(* CODESYS project oscat311.library
   Company: OSCAT
   Version: 3.11
   Author: www.oscat.de
   Title: LIBRARY

Project tree, tasks and I/O mapping:
  libraries: Standard, 3.3.1.10 (System)
  Data types/
    data type CALENDAR
    data type COMPLEX
    data type CONSTANTS_LANGUAGE
    data type CONSTANTS_LOCATION
    data type CONSTANTS_MATH
    data type CONSTANTS_PHYS
    data type CONSTANTS_SETUP
    data type ESR_DATA
    data type HOLIDAY_DATA
    data type NETWORK_BUFFER
    data type NETWORK_BUFFER_SHORT
    data type NW_BUF_LONG
    data type NW_BUF_SHORT
    data type REAL2
    data type SDT
    data type TIMER_EVENT
    data type URL
    data type VECTOR_3
  Global Variables/
    global variables Constants
    global variables Globale_Variablen
    global variables Setup_Data
  POUs/
    Buffer Management/
      function _BUFFER_CLEAR [ST]
      function _BUFFER_INIT [ST]
      function _BUFFER_INSERT [ST]
      function _STRING_TO_BUFFER [ST]
      function BUFFER_COMP [ST]
      function BUFFER_SEARCH [ST]
      function BUFFER_TO_STRING [ST]
    Building/
      actuators/
        function block ACTUATOR_2P [ST]
        function block ACTUATOR_3P [ST]
        function block ACTUATOR_A [ST]
        function block ACTUATOR_COIL [ST]
        function block ACTUATOR_PUMP [ST]
        function block ACTUATOR_UD [ST]
        function block AUTORUN [ST]
      electrical/
        function block CLICK [ST]
        function block CLICK_MODE [ST]
        function block DEBOUNCE [ST]
        function block DIMM_2 [ST]
        function block DIMM_I [ST]
        function block F_LAMP [ST]
        function block PULSE_LENGTH [ST]
        function block PULSE_T [ST]
        function block SW_RECONFIG [ST]
        function block SWITCH_I [ST]
        function block SWITCH_X [ST]
        function block TIMER_1 [ST]
        function block TIMER_2 [ST]
        function TIMER_EVENT_DECODE [ST]
        function block TIMER_EXT [ST]
        function block TIMER_P4 [ST]
      HLK/
        function AIR_DENSITY [ST]
        function AIR_ENTHALPY [ST]
        function block BOILER [ST]
        function block BURNER [ST]
        function DEW_CON [ST]
        function DEW_RH [ST]
        function DEW_TEMP [ST]
        function HEAT_INDEX [ST]
        function block HEAT_METER [ST]
        function block HEAT_TEMP [ST]
        function block LEGIONELLA [ST]
        function SDD [ST]
        function SDD_NH3 [ST]
        function SDT_NH3 [ST]
        function block T_AVG24 [ST]
        function block TEMP_EXT [ST]
        function WATER_CP [ST]
        function WATER_DENSITY [ST]
        function WATER_ENTHALPY [ST]
        function WCT [ST]
      Jalousie/
        function block BLIND_ACTUATOR [ST]
        function block BLIND_CONTROL [ST]
        function block BLIND_CONTROL_S [ST]
        function block BLIND_INPUT [ST]
        function block BLIND_NIGHT [ST]
        function block BLIND_SCENE [ST]
        function block BLIND_SECURITY [ST]
        function block BLIND_SET [ST]
        function block BLIND_SHADE [ST]
        function block BLIND_SHADE_S [ST]
    Device Drivers/
      function block IRTRANS_1 [ST]
      function block IRTRANS_4 [ST]
      function block IRTRANS_8 [ST]
      function block IRTRANS_DECODE [ST]
    Engineering/
      automation/
        function block DRIVER_1 [ST]
        function block DRIVER_4 [ST]
        function block DRIVER_4C [ST]
        function block FLOW_CONTROL [ST]
        function block FT_Profile [ST]
        function block INC_DEC [ST]
        function block INTERLOCK [ST]
        function block INTERLOCK_4 [ST]
        function MANUAL [ST]
        function block MANUAL_1 [ST]
        function block MANUAL_2 [ST]
        function block MANUAL_4 [ST]
        function block PARSET [ST]
        function block PARSET2 [ST]
        function block SIGNAL [ST]
        function block SIGNAL_4 [ST]
        function block SRAMP [ST]
        function block TANK_LEVEL [ST]
        function block TUNE [ST]
        function block TUNE2 [ST]
      control/
        function BAND_B [ST]
        function block CONTROL_SET1 [ST]
        function block CONTROL_SET2 [ST]
        function CTRL_IN [ST]
        function block CTRL_OUT [ST]
        function block CTRL_PI [ST]
        function block CTRL_PID [ST]
        function block CTRL_PWM [ST]
        function DEAD_BAND [ST]
        function block DEAD_BAND_A [ST]
        function DEAD_ZONE [ST]
        function block DEAD_ZONE2 [ST]
        function block FT_DERIV [ST]
        function block FT_IMP [ST]
        function block FT_INT [ST]
        function block FT_INT2 [ST]
        function block FT_PD [ST]
        function block FT_PDT1 [ST]
        function block FT_PI [ST]
        function block FT_PID [ST]
        function block FT_PIDW [ST]
        function block FT_PIDWL [ST]
        function block FT_PIW [ST]
        function block FT_PIWL [ST]
        function block FT_PT1 [ST]
        function block FT_PT2 [ST]
        function block FT_TN16 [ST]
        function block FT_TN64 [ST]
        function block FT_TN8 [ST]
        function block HYST [ST]
        function block HYST_1 [ST]
        function block HYST_2 [ST]
        function block HYST_3 [ST]
        function block INTEGRATE [ST]
      conversion/
        function block ASTRO [ST]
        function BFT_TO_MS [ST]
        function C_TO_F [ST]
        function C_TO_K [ST]
        function DEG_TO_DIR [ST]
        function DIR_TO_DEG [ST]
        function block ENERGY [ST]
        function F_TO_C [ST]
        function F_TO_OM [ST]
        function F_TO_PT [ST]
        function GEO_TO_DEG [ST]
        function K_TO_C [ST]
        function KMH_TO_MS [ST]
        function block LENGTH [ST]
        function MS_TO_BFT [ST]
        function MS_TO_KMH [ST]
        function OM_TO_F [ST]
        function block PRESSURE [ST]
        function PT_TO_F [ST]
        function block SPEED [ST]
        function block TEMPERATURE [ST]
      measurements/
        function block ALARM_2 [ST]
        function block BAR_GRAPH [ST]
        function block CALIBRATE [ST]
        function block CYCLE_TIME [ST]
        function block DT_SIMU [ST]
        function block M_D [ST]
        function block M_T [ST]
        function block M_TX [ST]
        function block METER [ST]
        function block METER_STAT [ST]
        function block ONTIME [ST]
        function T_PLC_MS [ST]
        function T_PLC_US [ST]
        function block TC_MS [ST]
        function block TC_S [ST]
        function block TC_US [ST]
      sensor/
        function MULTI_IN [ST]
        function RES_NI [ST]
        function RES_NTC [ST]
        function RES_PT [ST]
        function RES_SI [ST]
        function SENSOR_INT [ST]
        function TEMP_NI [ST]
        function TEMP_NTC [ST]
        function TEMP_PT [ST]
        function TEMP_SI [ST]
      signal generators/
        function block _RMP_B [ST]
        function block _RMP_NEXT [ST]
        function block _RMP_W [ST]
        function block GEN_PULSE [ST]
        function block GEN_PW2 [ST]
        function block GEN_RDM [ST]
        function block GEN_RDT [ST]
        function block GEN_RMP [ST]
        function block GEN_SIN [ST]
        function block GEN_SQR [ST]
        function block PWM_DC [ST]
        function block PWM_PW [ST]
        function block RMP_B [ST]
        function block RMP_SOFT [ST]
        function block RMP_W [ST]
      signal processing/
        function AIN [ST]
        function block AIN1 [ST]
        function AOUT [ST]
        function AOUT1 [ST]
        function BYTE_TO_RANGE [ST]
        function block DELAY [ST]
        function block DELAY_4 [ST]
        function block FADE [ST]
        function block FILTER_DW [ST]
        function block FILTER_I [ST]
        function block FILTER_MAV_DW [ST]
        function block FILTER_MAV_W [ST]
        function block FILTER_W [ST]
        function block FILTER_WAV [ST]
        function MIX [ST]
        function MUX_R2 [ST]
        function MUX_R4 [ST]
        function OFFSET [ST]
        function OFFSET2 [ST]
        function OVERRIDE [ST]
        function RANGE_TO_BYTE [ST]
        function RANGE_TO_WORD [ST]
        function SCALE [ST]
        function SCALE_B [ST]
        function SCALE_B2 [ST]
        function SCALE_B4 [ST]
        function SCALE_B8 [ST]
        function SCALE_D [ST]
        function SCALE_R [ST]
        function SCALE_X2 [ST]
        function SCALE_X4 [ST]
        function SCALE_X8 [ST]
        function block SEL2_OF_3 [ST]
        function block SEL2_OF_3B [ST]
        function block SH [ST]
        function block SH_1 [ST]
        function block SH_2 [ST]
        function block SH_T [ST]
        function STAIR [ST]
        function block STAIR2 [ST]
        function block TREND [ST]
        function block TREND_DW [ST]
        function WORD_TO_RANGE [ST]
    List Processing/
      function LIST_CLEAN [ST]
      function LIST_GET [ST]
      function LIST_INSERT [ST]
      function LIST_LEN [ST]
      function block LIST_NEXT [ST]
      function LIST_RETRIEVE [ST]
      function LIST_RETRIEVE_MAX [ST]
      function LIST_RETRIEVE_MIN [ST]
      function LIST_SORT_L [ST]
    Logic/
      FF edge triggered/
        function block COUNT_BR [ST]
        function block COUNT_DR [ST]
        function block FF_D2E [ST]
        function block FF_D4E [ST]
        function block FF_DRE [ST]
        function block FF_JKE [ST]
        function block FF_RSE [ST]
        function block SELECT_8 [ST]
        function block SHR_4E [ST]
        function block SHR_4UDE [ST]
        function block SHR_8PLE [ST]
        function block SHR_8UDE [ST]
        function block TOGGLE [ST]
      FF pulse triggered/
        function block LTCH [ST]
        function block LTCH_4 [ST]
        function block STORE_8 [ST]
      gate logic/
        function BCDC_TO_INT [ST]
        function BIT_COUNT [ST]
        function BIT_LOAD_B [ST]
        function BIT_LOAD_B2 [ST]
        function BIT_LOAD_DW [ST]
        function BIT_LOAD_DW2 [ST]
        function BIT_LOAD_W [ST]
        function BIT_LOAD_W2 [ST]
        function BIT_OF_DWORD [ST]
        function BIT_TOGGLE_B [ST]
        function BIT_TOGGLE_DW [ST]
        function BIT_TOGGLE_W [ST]
        function BYTE_OF_BIT [ST]
        function BYTE_OF_DWORD [ST]
        function block BYTE_TO_BITS [ST]
        function BYTE_TO_GRAY [ST]
        function CHECK_PARITY [ST]
        function block DEC_2 [ST]
        function block DEC_4 [ST]
        function block DEC_8 [ST]
        function DW_TO_REAL [ST]
        function DWORD_OF_BYTE [ST]
        function DWORD_OF_WORD [ST]
        function GRAY_TO_BYTE [ST]
        function INT_TO_BCDC [ST]
        function MUX_2 [ST]
        function MUX_4 [ST]
        function PARITY [ST]
        function REAL_TO_DW [ST]
        function REVERSE [ST]
        function SHL1 [ST]
        function SHR1 [ST]
        function SWAP_BYTE [ST]
        function SWAP_BYTE2 [ST]
        function WORD_OF_BYTE [ST]
        function WORD_OF_DWORD [ST]
      generators/
        function block A_TRIG [ST]
        function block B_TRIG [ST]
        function block CLICK_CNT [ST]
        function block CLICK_DEC [ST]
        function block CLK_DIV [ST]
        function block CLK_N [ST]
        function block CLK_PRG [ST]
        function block CLK_PULSE [ST]
        function block CYCLE_4 [ST]
        function block D_TRIG [ST]
        function block GEN_BIT [ST]
        function block GEN_SQ [ST]
        function block SCHEDULER [ST]
        function block SCHEDULER_2 [ST]
        function block SEQUENCE_4 [ST]
        function block SEQUENCE_64 [ST]
        function block SEQUENCE_8 [ST]
        function block TMAX [ST]
        function block TMIN [ST]
        function block TOF_1 [ST]
        function block TONOF [ST]
        function block TP_1 [ST]
        function block TP_1D [ST]
        function block TP_X [ST]
      memory/
        function block FIFO_16 [ST]
        function block FIFO_32 [ST]
        function block STACK_16 [ST]
        function block STACK_32 [ST]
      Others/
        function CRC_CHECK [ST]
        function CRC_GEN [ST]
        function block MATRIX [ST]
        function block PIN_CODE [ST]
    Mathematical/
      Array/
        function _ARRAY_ABS [ST]
        function _ARRAY_ADD [ST]
        function _ARRAY_INIT [ST]
        function _ARRAY_MEDIAN [ST]
        function _ARRAY_MUL [ST]
        function _ARRAY_SHUFFLE [ST]
        function _ARRAY_SORT [ST]
        function ARRAY_AVG [ST]
        function ARRAY_GAV [ST]
        function ARRAY_HAV [ST]
        function ARRAY_MAX [ST]
        function ARRAY_MIN [ST]
        function ARRAY_SDV [ST]
        function ARRAY_SPR [ST]
        function ARRAY_SUM [ST]
        function ARRAY_TREND [ST]
        function ARRAY_VAR [ST]
        function IS_SORTED [ST]
      Complex/
        function CABS [ST]
        function CACOS [ST]
        function CACOSH [ST]
        function CADD [ST]
        function CARG [ST]
        function CASIN [ST]
        function CASINH [ST]
        function CATAN [ST]
        function CATANH [ST]
        function CCON [ST]
        function CCOS [ST]
        function CCOSH [ST]
        function CDIV [ST]
        function CEXP [ST]
        function CINV [ST]
        function CLOG [ST]
        function CMUL [ST]
        function CPOL [ST]
        function CPOW [ST]
        function CSET [ST]
        function CSIN [ST]
        function CSINH [ST]
        function CSQRT [ST]
        function CSUB [ST]
        function CTAN [ST]
        function CTANH [ST]
      Double Precision/
        function R2_ABS [ST]
        function R2_ADD [ST]
        function R2_ADD2 [ST]
        function R2_MUL [ST]
        function R2_SET [ST]
      functions/
        function F_LIN [ST]
        function F_LIN2 [ST]
        function F_POLY [ST]
        function F_POWER [ST]
        function F_QUAD [ST]
        function block FT_AVG [ST]
        function block FT_MIN_MAX [ST]
        function block FT_RMP [ST]
        function LINEAR_INT [ST]
        function POLYNOM_INT [ST]
      Geometry/
        function CIRCLE_A [ST]
        function CIRCLE_C [ST]
        function CONE_V [ST]
        function ELLIPSE_A [ST]
        function ELLIPSE_C [ST]
        function SPHERE_V [ST]
        function TRIANGLE_A [ST]
      Vektormathematik/
        function V3_ABS [ST]
        function V3_ADD [ST]
        function V3_ANG [ST]
        function V3_DPRO [ST]
        function V3_NORM [ST]
        function V3_NUL [ST]
        function V3_PAR [ST]
        function V3_REV [ST]
        function V3_SMUL [ST]
        function V3_SUB [ST]
        function V3_XANG [ST]
        function V3_XPRO [ST]
        function V3_YANG [ST]
        function V3_ZANG [ST]
      function ACOSH [ST]
      function ACOTH [ST]
      function AGDF [ST]
      function ASINH [ST]
      function ATAN2 [ST]
      function ATANH [ST]
      function BETA [ST]
      function BINOM [ST]
      function CAUCHY [ST]
      function CAUCHYCD [ST]
      function CEIL [ST]
      function CEIL2 [ST]
      function CMP [ST]
      function COSH [ST]
      function COTH [ST]
      function D_TRUNC [ST]
      function DEC1 [ST]
      function DEG [ST]
      function DIFFER [ST]
      function ERF [ST]
      function ERFC [ST]
      function EVEN [ST]
      function EXP10 [ST]
      function EXPN [ST]
      function FACT [ST]
      function FIB [ST]
      function FLOOR [ST]
      function FLOOR2 [ST]
      function FRACT [ST]
      function GAMMA [ST]
      function GAUSS [ST]
      function GAUSSCD [ST]
      function GDF [ST]
      function GOLD [ST]
      function HYPOT [ST]
      function INC [ST]
      function INC1 [ST]
      function INC2 [ST]
      function INV [ST]
      function LAMBERT_W [ST]
      function LANGEVIN [ST]
      function MAX3 [ST]
      function MID3 [ST]
      function MIN3 [ST]
      function MODR [ST]
      function MUL_ADD [ST]
      function NEGX [ST]
      function RAD [ST]
      function RDM [ST]
      function RDM2 [ST]
      function RDMDW [ST]
      function RND [ST]
      function ROUND [ST]
      function SGN [ST]
      function SIGMOID [ST]
      function SIGN_I [ST]
      function SIGN_R [ST]
      function SINC [ST]
      function SINH [ST]
      function SQRTN [ST]
      function TANC [ST]
      function TANH [ST]
      function WINDOW [ST]
      function WINDOW2 [ST]
    Network/
      function HTML_DECODE [ST]
      function HTML_ENCODE [ST]
      function IP4_CHECK [ST]
      function IP4_DECODE [ST]
      function IP4_TO_STRING [ST]
      function IS_IP4 [ST]
      function IS_URLCHR [ST]
      function STRING_TO_URL [ST]
      function URL_DECODE [ST]
      function URL_ENCODE [ST]
      function URL_TO_STRING [ST]
    Other/
      function block ESR_COLLECT [ST]
      function block ESR_MON_B8 [ST]
      function block ESR_MON_R4 [ST]
      function block ESR_MON_X8 [ST]
      function OSCAT_VERSION [ST]
      function STATUS_TO_ESR [ST]
    String/
      function BIN_TO_BYTE [ST]
      function BIN_TO_DWORD [ST]
      function BYTE_TO_STRB [ST]
      function BYTE_TO_STRH [ST]
      function CAPITALIZE [ST]
      function CHARCODE [ST]
      function CHARNAME [ST]
      function CHR_TO_STRING [ST]
      function CLEAN [ST]
      function CODE [ST]
      function COUNT_CHAR [ST]
      function DEC_TO_BYTE [ST]
      function DEC_TO_DWORD [ST]
      function DEC_TO_INT [ST]
      function DEL_CHARS [ST]
      function DT_TO_STRF [ST]
      function DWORD_TO_STRB [ST]
      function DWORD_TO_STRF [ST]
      function DWORD_TO_STRH [ST]
      function EXEC [ST]
      function FILL [ST]
      function FIND_CHAR [ST]
      function FIND_CTRL [ST]
      function FIND_NONUM [ST]
      function FIND_NUM [ST]
      function FINDB [ST]
      function FINDB_NONUM [ST]
      function FINDB_NUM [ST]
      function FINDP [ST]
      function FIX [ST]
      function FLOAT_TO_REAL [ST]
      function FSTRING_TO_BYTE [ST]
      function FSTRING_TO_DT [ST]
      function FSTRING_TO_DWORD [ST]
      function FSTRING_TO_MONTH [ST]
      function FSTRING_TO_WEEK [ST]
      function FSTRING_TO_WEEKDAY [ST]
      function HEX_TO_BYTE [ST]
      function HEX_TO_DWORD [ST]
      function IS_ALNUM [ST]
      function IS_ALPHA [ST]
      function IS_CC [ST]
      function IS_CTRL [ST]
      function IS_HEX [ST]
      function IS_LOWER [ST]
      function IS_NCC [ST]
      function IS_NUM [ST]
      function IS_UPPER [ST]
      function ISC_ALPHA [ST]
      function ISC_CTRL [ST]
      function ISC_HEX [ST]
      function ISC_LOWER [ST]
      function ISC_NUM [ST]
      function ISC_UPPER [ST]
      function LOWERCASE [ST]
      function block MESSAGE_4R [ST]
      function block MESSAGE_8 [ST]
      function MIRROR [ST]
      function MONTH_TO_STRING [ST]
      function OCT_TO_BYTE [ST]
      function OCT_TO_DWORD [ST]
      function REAL_TO_STRF [ST]
      function REPLACE_ALL [ST]
      function REPLACE_CHARS [ST]
      function REPLACE_UML [ST]
      function block TICKER [ST]
      function TO_LOWER [ST]
      function TO_UML [ST]
      function TO_UPPER [ST]
      function TRIM [ST]
      function TRIM1 [ST]
      function TRIME [ST]
      function UPPERCASE [ST]
      function WEEKDAY_TO_STRING [ST]
    Time&Date/
      function block CALENDAR_CALC [ST]
      function DATE_ADD [ST]
      function DAY_OF_DATE [ST]
      function DAY_OF_MONTH [ST]
      function DAY_OF_WEEK [ST]
      function DAY_OF_YEAR [ST]
      function DAY_TO_TIME [ST]
      function DAYS_DELTA [ST]
      function DAYS_IN_MONTH [ST]
      function DAYS_IN_YEAR [ST]
      function block DCF77 [ST]
      function DST [ST]
      function DT_TO_SDT [ST]
      function DT2_TO_SDT [ST]
      function EASTER [ST]
      function block HOLIDAY [ST]
      function HOUR [ST]
      function HOUR_OF_DT [ST]
      function HOUR_TO_TIME [ST]
      function HOUR_TO_TOD [ST]
      function JD2000 [ST]
      function LEAP_DAY [ST]
      function LEAP_OF_DATE [ST]
      function LEAP_YEAR [ST]
      function LTIME_TO_UTC [ST]
      function MINUTE [ST]
      function MINUTE_OF_DT [ST]
      function MINUTE_TO_TIME [ST]
      function MONTH_BEGIN [ST]
      function MONTH_END [ST]
      function MONTH_OF_DATE [ST]
      function MULTIME [ST]
      function PERIOD [ST]
      function PERIOD2 [ST]
      function REFRACTION [ST]
      function block RTC_2 [ST]
      function block RTC_MS [ST]
      function SDT_TO_DATE [ST]
      function SDT_TO_DT [ST]
      function SDT_TO_TOD [ST]
      function SECOND [ST]
      function SECOND_OF_DT [ST]
      function SECOND_TO_TIME [ST]
      function SET_DATE [ST]
      function SET_DT [ST]
      function SET_TOD [ST]
      function block SUN_POS [ST]
      function block SUN_TIME [ST]
      function TIMECHECK [ST]
      function UTC_TO_LTIME [ST]
      function WORK_WEEK [ST]
      function YEAR_BEGIN [ST]
      function YEAR_END [ST]
      function YEAR_OF_DATE [ST]
  Visualizations/
*)

// Data types/CALENDAR
TYPE CALENDAR :
STRUCT
	UTC : DT;						(* world time UTC *)
	LDT : DT;						(* local time *)
	LDATE : DATE;				(* local date *)
	LTOD : TOD;					(* local time of day *)
	YEAR : INT;					(* year of LDATE *)
	MONTH : INT;					(* month of LDATE *)
	DAY : INT;						(* day of LDATE *)
	WEEKDAY : INT;				(* weekday of LDATE *)
	OFFSET : INT;					(* Time Zone Offset for Local time in minutes *)
	DST_EN : BOOL;				(* daylight savings time enable *)
	DST_ON : BOOL;				(* true when daylight savings time os on *)
	NAME : STRING(5);			(* name of time zone *)
	LOCATION : INT;				(* location number pls see location setup *)
	LONGITUDE : REAL;			(* longitude of current location *)
	LATITUDE : REAL;			(* latitude of current location *)
	SUN_RISE : TOD;				(* sun_rise for current location *)
	SUN_SET : TOD;				(* sun_set for current location *)
	SUN_MIDDAY : TOD;			(* worldtime when sun stands at south position *)
	SUN_HEIGTH : REAL	;		(* suns heigth at midday, south position *)
	SUN_HOR : REAL;			(* sun angle horizontal 0 = north in degrees *)
	SUN_VER : REAL;			(* sun angle vertical above horizon in degrees *)
	NIGHT : BOOL;				(* true between sun_set and sun_rise *)
	HOLIDAY : BOOL;				(* true when holiday *)
	HOLY_NAME : STRING(30);	(* name of holiday *)
	WORK_WEEK : INT;			(* current work week *)
END_STRUCT
END_TYPE

// Data types/COMPLEX
TYPE COMPLEX :
STRUCT
	re : REAL;
	im : REAL;
END_STRUCT
END_TYPE

// Data types/CONSTANTS_LANGUAGE
TYPE CONSTANTS_LANGUAGE :
STRUCT
	(* Language Setup *)
	DEFAULT : INT := 1; (* 1=english, 2=german 3=french *)
	LMAX : INT := 3;
	WEEKDAYS : ARRAY[1..3, 1..7] OF STRING(10) :=[	'Monday', 'Tuesday', 'Wednesday', 'Thursday', 'Friday', 'Saturday', 'Sunday',
													'Montag', 'Dienstag', 'Mittwoch', 'Donnerstag', 'Freitag', 'Samstag', 'Sonntag',
													'Lundi', 'Mardi', 'Mercredi', 'Jeudi', 'Vendredi', 'Samedi', 'Dimanche'];
	WEEKDAYS2 : ARRAY[1..3, 1..7] OF STRING(2) :=[	'Mo', 'Tu', 'We', 'Th', 'Fr', 'Sa', 'Su',
													'Mo', 'Di', 'Mi', 'Do', 'Fr', 'Sa', 'So',
													'Lu', 'Ma', 'Me', 'Je', 'Ve', 'Sa', 'Di'];
	MONTHS : ARRAY[1..3, 1..12] OF STRING(10) :=[	'January', 'February', 'March', 'April', 'May', 'June', 'July', 'August', 'September', 'October', 'November', 'December',
													'Januar', 'Februar', 'März', 'April', 'Mai', 'Juni', 'Juli', 'August', 'September', 'Oktober', 'November', 'Dezember',
													'Janvier', 'Février', 'mars', 'Avril', 'Mai', 'Juin', 'Juillet', 'Août', 'Septembre', 'Octobre', 'Novembre', 'Decembre'];
	MONTHS3 : ARRAY[1..3, 1..12] OF STRING(3) :=[	'Jan', 'Feb', 'Mar', 'Apr', 'May', 'Jun', 'Jul', 'Aug', 'Sep', 'Oct', 'Nov', 'Dec',
													'Jan', 'Feb', 'Mrz', 'Apr', 'Mai', 'Jun', 'Jul', 'Aug', 'Sep', 'Okt', 'Nov', 'Dez',
													'Jan', 'Fev', 'Mar', 'Avr', 'Mai', 'Jun', 'Jul', 'Aou', 'Sep', 'Oct', 'Nov', 'Dec'];
	DIRS : ARRAY[1..3,0..15] OF STRING(3) :=[		'N', 'NNE', 'NE', 'ENE', 'E', 'ESE', 'SE', 'SSE', 'S', 'SSW', 'SW', 'WSW', 'W', 'WNW', 'NW', 'NNW',
													'N', 'NNO', 'NO', 'ONO', 'O', 'OSO', 'SO', 'SSO', 'S', 'SSW', 'SW', 'WSW', 'W', 'WNW', 'NW', 'NNW',
													'N', 'NNO', 'NO', 'ONO', 'O', 'OSO', 'SO', 'SSO', 'S', 'SSW', 'SW', 'WSW', 'W', 'WNW', 'NW', 'NNW'];
END_STRUCT
END_TYPE

// Data types/CONSTANTS_LOCATION
TYPE CONSTANTS_LOCATION :
STRUCT
	(* location setup *)
	DEFAULT : INT := 1; (* 1=germany, 2=austria 3=france *)
	LMAX : INT := 3;

	(*	if month = 0 then F_day is the offset in days from easter
		used :0 = NOT used, 1 = used, -1..-7 menas the weekday before the specified DATE example -3 means wednesday before 23.11
	*)
	HOLIDAY : ARRAY[1..3, 0..29] OF HOLIDAY_DATA :=[ (name := 'Neujahr', day := 1, month := 1, use := 1),
													(name := 'Heilig Drei Könige', day := 6, month := 1, use := 1),
													(name := 'Karfreitag', day := -2, month := 0, use := 1),
													(name := 'Ostersonntag', day := 0, month := 0, use := 1),
													(name := 'Ostermontag', day := 1, month := 0, use := 1),
													(name := 'Tag der Arbeit', day := 1, month := 5, use := 1),
													(name := 'Christi Himmelfahrt', day := 39, month := 0, use := 1),
													(name := 'Pfingstsonntag', day := 49, month := 0, use := 1),
													(name := 'Pfingstmontag', day := 50, month := 0, use := 1),
													(name := 'Fronleichnam', day := 60, month := 0, use := 1),
													(name := 'Augsburger Friedensfest', day := 8, month := 8, use := 0),
													(name := 'Maria Himmelfahrt', day := 15, month := 8, use := 1),
													(name := 'Tag der Deutschen Einheit', day := 3, month := 10, use := 1),
													(name := 'Reformationstag', day := 31, month := 10, use := 0),
													(name := 'Allerheiligen', day := 1, month := 11, use := 1),
													(name := 'Buss und Bettag', day := 23, month := 11, use := 0),
													(name := '1. Weihnachtstag', day := 25, month := 12, use := 1),
													(name := '2. Weihnachtstag', day := 26, month := 12, use := 1),
													(),
													(),
													(),
													(),
													(),
													(),
													(),
													(),
													(),
													(),
													(),
													(),
													(* the next 30 lines are for austrian holidays *)
													(name := 'Neujahr', day := 1, month := 1, use := 1),
													(name := 'Heilig Drei Könige', day := 6, month := 1, use := 1),
													(name := 'Karfreitag', day := -2, month := 0, use := 1),
													(name := 'Ostersonntag', day := 0, month := 0, use := 1),
													(name := 'Ostermontag', day := 1, month := 0, use := 1),
													(name := '', day := 1, month := 5, use := 0),
													(name := 'Christi Himmelfahrt', day := 39, month := 0, use := 1),
													(name := 'Pfingstsonntag', day := 49, month := 0, use := 1),
													(name := 'Pfingstmontag', day := 50, month := 0, use := 1),
													(name := 'Fronleichnam', day := 60, month := 0, use := 1),
													(name := '', day := 8, month := 8, use := 0),
													(name := 'Maria Himmelfahrt', day := 15, month := 8, use := 1),
													(name := '', day := 3, month := 10, use := 0),
													(name := '', day := 31, month := 10, use := 0),
													(name := 'Allerheiligen', day := 1, month := 11, use := 1),
													(name := 'Maria Empfängnis', day := 8, month := 12, use := 1),
													(name := '1. Weihnachtstag', day := 25, month := 12, use := 1),
													(name := '2. Weihnachtstag', day := 26, month := 12, use := 1),
													(),
													(),
													(),
													(),
													(),
													(),
													(),
													(),
													(),
													(),
													(),
													(),
													(* the next 30 lines are for french holidays *)
													(name := 'Nouvel an', day := 1, month := 1, use := 1),
													(name := 'St Valentin', day := 14, month := 2, use := 0),
													(name := 'Vendredi Saint (alsace)', day := -2, month := 0, use := 0),
													(name := 'Dimanche de pâques', day := 0, month := 0, use := 1),
													(name := 'Lundi de pâques', day := 1, month := 0, use := 1),
													(name := 'Jeudi de Ascension', day := 39, month := 0, use := 1),
													(name := 'dimanche de Pentecôte ', day := 49, month := 0, use := 1),
													(name := 'jeudi de la Trinité', day := 60, month := 0, use := 0),
													(name := 'Fête du travail', day := 1, month := 5, use := 1),
													(name := 'Victoire 1945 ', day := 8, month := 5, use := 1),
													(name := 'Prise de La bastille', day := 14, month := 7, use := 1),
													(name := '15 Août 1944', day := 15, month := 8, use := 1),
													(name := 'Halloween', day := 31, month := 10, use := 0),
													(name := 'Armistice 1918', day := 11, month := 11, use := 1),
													(name := 'Noël', day := 25, month := 12, use := 1),
													(name := 'Saint Étienne (alsace)', day := 26, month := 12, use := 0),
													(name := 'Fête de la musique', day := 21, month := 6, use := 0),
													(),
													(),
													(),
													(),
													(),
													(),
													(),
													(),
													(),
													(),
													(),
													(),
													()];

END_STRUCT
END_TYPE

// Data types/CONSTANTS_MATH
TYPE CONSTANTS_MATH :
STRUCT
	PI : REAL := 	3.14159265358979323846264338327950288;	(* Kreiszahl PI *)
	PI2 : REAL := 	6.28318530717958647692528676655900576;	(* PI * 2 *)
	PI4 : REAL :=  12.56637061435917295385057353311801152;	(* PI * 4 *)
	PI05 : REAL :=  1.5707963267949;						(* PI / 2 *)
	PI025 : REAL := 0.785398163397448;						(* PI / 4 *)
	PI_INV : REAL := 0.318309886183791;						(* 1 / PI *)
	E : REAL := 	2.71828182845904523536028747135266249;	(* Eulersche Konstante e *)
	E_INV : REAL := 0.367879441171442;						(* 1 / e *)
	SQ2 : REAL :=	1.4142135623731;						(* Wurzel von 2 *)
END_STRUCT
END_TYPE

// Data types/CONSTANTS_PHYS
TYPE CONSTANTS_PHYS :
STRUCT
	C : REAL := 299792458.0;				(* Lichtgeschwindigkeit in m/s *)
	E : REAL := 1.60217653E-19;				(* elementarladung in Colomb = A * s *)
	G : REAL := 9.80665; 						(* Erdbeschleunigung in m / s² *)
	T0 : REAL := -273.15;						(* absoluter Nullpunkt in °C *)
	RU : REAL := 8.314472; 					(* Universelle Gaskonstante in J / (mol · K) *)
	PN : REAL := 101325.0;					(* NormalDruck in Pa *)
END_STRUCT
END_TYPE

// Data types/CONSTANTS_SETUP
TYPE CONSTANTS_SETUP :
STRUCT
	(* setup Parameters *)
	EXTENDED_ASCII : BOOL := TRUE;
	CHARNAMES : ARRAY[1..4] OF STRING(253) :=[ ';"&quot;&&amp;<&lt;>&gt;&euro; &nbsp;¡&iexcl;¢&cent;£&pound;¤&curren;¥&yen;¦&brvbar;§&sect;¨&uml;©&copy;ª&ordf;«&laquo;¬&not;­&shy;®&reg;¯&macr;°&deg;±&plusmn;²&sup2;³&sup3;´&acute;µ&micro;¶&para;·&middot;¸&cedil;¹&sup1;º&ordm;»&raquo;¼&frac14;Û&Ucirc;',
		';¾&frac34;¿&iquest;À&Agrave;Á&Aacute;Â&Acirc;Ã&Atilde;Ä&Auml;Å&Aring;Æ&AElig;Ç&Ccedil;È&Egrave;É&Eacute;Ê&Ecirc;Ë&Euml;Ì&Igrave;Í&Iacute;Î&Icirc;Ï&Iuml;Ð&ETH;Ñ&Ntilde;Ò&Ograve;Ó&Oacute;Ô&Ocirc;Õ&Otilde;Ö&Ouml;×&times;Ø&Oslash;Ù&Ugrave;Ú&Uacute;½&frac12;',
		';Ü&Uuml;Ý&Yacute;Þ&THORN;ß&szlig;à&agrave;á&aacute;â&acirc;ã&atilde;ä&auml;å&aring;æ&aelig;ç&ccedil;è&egrave;é&eacute;ê&ecirc;ë&euml;ì&igrave;í&iacute;î&icirc;ï&iuml;ð&eth;ñ&ntilde;ò&ograve;ó&oacute;ô&ocirc;õ&otilde;ö&ouml;÷&divide;ø&oslash;ù&ugrave;',
		';ú&uacute;û&ucirc;ü&uuml;ý&yacute;þ&thorn;ÿ&yuml;'];
	MTH_OFS : ARRAY[1..12] OF INT :=[ 0,31,59,90,120,151,181,212,243,273,304,334];
	DECADES : ARRAY[0..8] OF REAL :=[ 1,10,100,1000,10000,10000,100000,1000000,10000000];
END_STRUCT
END_TYPE

// Data types/ESR_DATA
TYPE ESR_DATA :
STRUCT
	TYP : BYTE;
	ADRESS : STRING(10);
	DS : DT;
	TS : TIME;
	DATA : ARRAY[0..7] OF BYTE;
END_STRUCT
END_TYPE

// Data types/HOLIDAY_DATA
TYPE HOLIDAY_DATA :
STRUCT
	NAME : STRING(30);
	DAY : SINT;
	MONTH : SINT;
	USE : SINT;
END_STRUCT
END_TYPE

// Data types/NETWORK_BUFFER
TYPE NETWORK_BUFFER :
STRUCT
	SIZE : UINT;
	BUFFER : NW_BUF_LONG;
END_STRUCT
END_TYPE

// Data types/NETWORK_BUFFER_SHORT
TYPE NETWORK_BUFFER_SHORT :
STRUCT
	SIZE : UINT;
	BUFFER : NW_BUF_SHORT;
END_STRUCT
END_TYPE

// Data types/NW_BUF_LONG
TYPE
	NW_BUF_LONG  : ARRAY[0..NETWORK_BUFFER_LONG_SIZE] OF BYTE;
END_TYPE

// Data types/NW_BUF_SHORT
TYPE
	NW_BUF_SHORT : ARRAY[0..NETWORK_BUFFER_SHORT_SIZE] OF BYTE;
END_TYPE

// Data types/REAL2
TYPE REAL2 :
STRUCT
	R1 : REAL;	(* small value *)
	RX : REAL;	(* big value *)
END_STRUCT
END_TYPE

// Data types/SDT
TYPE SDT :
STRUCT
	YEAR : INT;
	MONTH : INT;
	DAY : INT;
	WEEKDAY : INT;
	HOUR : INT;
	MINUTE : INT;
	SECOND : INT;
	MS : INT;
END_STRUCT
END_TYPE

// Data types/TIMER_EVENT
TYPE TIMER_EVENT :
STRUCT
	TYP : BYTE;
	CHANNEL : BYTE;
	DAY : BYTE;
	START : TOD;
	DURATION : TIME;
	LAND : BYTE;
	LOR : BYTE;
	LAST : DWORD;
END_STRUCT
END_TYPE

// Data types/URL
TYPE URL :
STRUCT
	PROTOCOL : STRING(10);
	USER : STRING(20);
	PASSWORD : STRING(20);
	DOMAIN : STRING(80);
	PORT : WORD;
	PATH : STRING(80);
	QUERY : STRING(40);
	ANCHOR : STRING(40);
END_STRUCT
END_TYPE

// Data types/VECTOR_3
TYPE VECTOR_3 :
STRUCT
	X : REAL;
	Y : REAL;
	Z : REAL;
END_STRUCT
END_TYPE

// Global Variables/Constants
VAR_GLOBAL CONSTANT
	STRING_LENGTH : INT := 250;
	NETWORK_BUFFER_LONG_SIZE : UINT := 3999;
	NETWORK_BUFFER_SHORT_SIZE : UINT := 1459;
END_VAR




(* revisionhistory
hm 3. mar. 2007
	extended accuracy of pi2
	renamed T0 to Tk for better compatibility with other libraries
	renamed C t0 c0 for better compatibility

hm	2. may. 2007
	added RU universal gas constant

hm	1. oct. 2007
	added setup parameter STEP7

hm 31. oct. 2007
	added PN

hm	6. mar. 2008
	added setup Parameter EXTENDED_ASCII

hm	28. Mar. 2008
	added setup parameter STRING_LENGTH

hm	7. apr. 2008
	Deleted unused setup parameter Step7

hm	19. apr. 2008
	added setup parameter NETWORK_BUFFER_SIZE

hm	27. apr. 2008
	added PI05 and PI025

hm	18. may. 2008
	added charname lists
	renamed E to E1

hm	30. jun. 2008
	reduced size of string constants to 253 to avoid problems with target aixia DCUF

hm	21. sep. 2008
	added section language setup
	added section location setup

hm	20. oct. 2008
	changed to structured constants

hm	16. nov. 2008
	moved structured constants to global vars for compatibility reasons

hm	13. nov. 2009
	added network_buffer_short_size
	renamed network_buffer_long_size
	changed string length to 250
*)

// Global Variables/Globale_Variablen
VAR_GLOBAL
	MATH : CONSTANTS_MATH;
	PHYS : CONSTANTS_PHYS;
	LANGUAGE : CONSTANTS_LANGUAGE;
	SETUP : CONSTANTS_SETUP;
	LOCATION : CONSTANTS_LOCATION;
END_VAR

// Global Variables/Setup_Data
VAR_GLOBAL RETAIN

END_VAR

// POUs/Mathematical/Array/_ARRAY_ABS
FUNCTION _ARRAY_ABS : BOOL
VAR_INPUT
	pt : POINTER TO ARRAY[0..32000] OF REAL;
	size : UINT;
END_VAR
VAR
	i: UINT;
	stop: UINT;
END_VAR

(*
version 1.0	2. apr. 2008
programmer 	hugo
tested by	tobias

this function will calculate the absolute value of each element of the array and stroe the result instead of the element.
Array[i] := ABS(ARRAY[i]).
the function needs to be called:	array_avg(adr("array"),sizeof("array"));
because this function works with pointers its very time efficient and it needs no extra memory.

*)

stop := SHR(size,2)-1;
FOR i := 0 TO stop DO
	PT^[i] := ABS(PT^[i]);
END_FOR;
_ARRAY_ABS := TRUE;


(* revision history
hm	2. apr 2008		rev 1.0
	original version

*)

END_FUNCTION

// POUs/Mathematical/Array/ARRAY_AVG
FUNCTION ARRAY_AVG : REAL
VAR_INPUT
	pt : POINTER TO ARRAY[0..32000] OF REAL;
	size : UINT;
END_VAR
VAR
	i: UINT;
	stop: UINT;
END_VAR

(*
version 1.3	10. mar. 2009
programmer 	hugo
tested by		tobias

this function will calculate the average of a given array.
the function needs to be called:	array_avg(adr("array"),sizeof("array"));
because this function works with pointers its very time efficient and it needs no extra memory.

*)

stop := SHR(size,2)-1;
ARRAY_AVG := pt^[0];
FOR i := 1 TO stop DO
	ARRAY_AVG := ARRAY_AVG + pt^[i];
END_FOR;
ARRAY_AVG := ARRAY_AVG / UINT_TO_REAL(stop + 1);


(* revision history
hm	2. oct 2007		rev 1.0
	original version

hm	12. dec 2007	rev 1.1
	chaged code for better performance

hm	16. mar. 2008	rev 1.2
	changed input size to uint

hm	10. mar. 2009	rev 1.3
	added type conversion for compatibility reasons
*)

END_FUNCTION

// POUs/String/CODE
FUNCTION CODE : BYTE
VAR_INPUT
	STR : STRING(STRING_LENGTH);
	POS : INT;
END_VAR
VAR
	PT : POINTER TO BYTE;
END_VAR

(*
version 1.1	29. mar. 2008
programmer 	hugo
tested by		tobias

code extracts the code of a character at position POS of a string STR.

*)

IF pos < 1 OR pos > LEN(str) THEN
	CODE := 0;
	RETURN;
ELSE
	PT := ADR(STR) + INT_TO_DWORD(pos - 1);
	CODE := pt^;
END_IF;

(* revision history
hm	9. mar. 2008	rev 1.0
	original version

hm	29. mar. 2008	rev 1.1
	changed STRING to STRING(STRING_LENGTH)
*)

END_FUNCTION

// POUs/Mathematical/Array/_ARRAY_ADD
FUNCTION _ARRAY_ADD : BOOL
VAR_INPUT
	pt : POINTER TO ARRAY[0..32000] OF REAL;
	size : UINT;
	X : REAL;
END_VAR
VAR
	i: UINT;
	stop: UINT;
END_VAR

(*
version 1.0	2. apr. 2008
programmer 	hugo
tested by	tobias

this function will add an offset X to each element of the array and stroe the result instead of the element.
Array[i] := ARRAY[i] + X.
the function needs to be called:	array_avg(adr("array"),sizeof("array"));
because this function works with pointers its very time efficient and it needs no extra memory.

*)

stop := SHR(size,2)-1;
FOR i := 0 TO stop DO
	PT^[i] := PT^[i] + X;
END_FOR;
_ARRAY_ADD := TRUE;


(* revision history
hm	2. apr 2008		rev 1.0
	original version

*)

END_FUNCTION

// POUs/Engineering/signal processing/OFFSET
FUNCTION OFFSET : REAL
VAR_INPUT
	X : REAL;
	O1, O2, O3, O4 : BOOL;
	D : BOOL;
END_VAR
VAR_INPUT CONSTANT
	Offset_1 : REAL;
	Offset_2 : REAL;
	Offset_3 : REAL;
	Offset_4 : REAL;
	default : REAL;
END_VAR

(*
version 1.0	12 jan 2007
programmer 	oscat
tested by	oscat

The Function offset adds offsets to an analog signal depending on digital inputs.
all selected offsets are added at the same time.
with the input D a default value instead of the input X can be used.

*)

IF D THEN OFFSET := default; ELSE OFFSET := X; END_IF;
IF O1 THEN OFFSET := OFFSET + offset_1; END_IF;
IF O2 THEN OFFSET := OFFSET + offset_2; END_IF;
IF O3 THEN OFFSET := OFFSET + offset_3; END_IF;
IF O4 THEN OFFSET := OFFSET + offset_4; END_IF;



(* revision history
hm	12. jan 2007
	original version


*)

END_FUNCTION

// POUs/Engineering/automation/SIGNAL
FUNCTION_BLOCK SIGNAL
VAR_INPUT
	IN : BOOL;
	SIG : BYTE;
	TS : TIME;
END_VAR
VAR_OUTPUT
	Q : BOOL;
END_VAR
VAR
	tx: DWORD;
	step: BYTE;
END_VAR
VAR CONSTANT
	one : BYTE := 1;
END_VAR

(*
version 1.0	13 dec 2007
programmer 	hugo
tested by		tobias

this function generates an output signal according to a bit pattern SIG.
the patter is shifted to the output in time steps of TS.
ts defaults to 128 ms if not specified.
*)

IF in THEN
	(* an alarm is present read system time first *)
	tx := T_PLC_MS();
	(* calculate the step counter which is the lowest 3 bits of (time / ts) *)
	IF ts > t#0s THEN
		step := DWORD_TO_BYTE(tx / TIME_TO_DWORD(ts) AND 16#0000_0007);
	ELSE
		step := DWORD_TO_BYTE(SHR(tx,7) AND 16#0000_0007);
	END_IF;
	(* convert the value 0-7 in step into one bit only (bit 0-7) *)
	step := SHL(one,step);
	(* generate the output signal *)
	Q := (step AND sig) > 0;
ELSE
	Q := FALSE;
END_IF;

(* revision history
hm	13.12.2007		rev 1.0
	original version

*)

END_FUNCTION_BLOCK

// POUs/Engineering/measurements/T_PLC_MS
FUNCTION T_PLC_MS : DWORD
VAR CONSTANT
	debug : BOOL := 0;
	N : INT := 0;
	offset : DWORD := 0;
END_VAR
VAR
	tx : TIME;
END_VAR

(*
version 1.2	16. nov 2008
programmer 	hugo
tested by	oscat

T_PLC_MS reads the internal PLC timer and return the time, it has the advantage to be able to set a debug mode 
and speed up the counter to test the plc timer overrun which occurs every 50 days respectively 25 days at siemens S7
this routine also allows to correct the behavior of s7 where the internal plc counter will not count all 32 bits.

*)

tx := TIME();
T_PLC_MS := TIME_TO_DWORD(Tx);
(* hier muss die korrektur für step7 stattfinden
plctime muss den vollen wertebereich von time ausnutzen:
wenn bei step7 time -24tage bis plus 24 tage ist dann muss der timer auch beim überlauf auf -24tage springen 
und auf keinen fall auf 0 !!!!
für siemens muss ein weiterer fb im main eingebunden werden der sicherstellt das alle 32 bits durchgezählt werden.
es kann nur ein fb sein den er muss sich das oberste (32te) bit merken.
oder etwa spring s7 bei überlauf auf -24 tage????? dann wäre keine korrektur nötig.
*)
IF debug THEN
	T_PLC_MS := (SHL(T_PLC_MS,N) OR SHL(DWORD#1,N)-1) + OFFSET;
END_IF;

(* revision history
hm	14.9.2007	rev 1.0
	original version

hm	12. nov 2007	rev 1.1
	added temporaray variable tx because some compilers could not handle time() as an argument

hm	16. nov. 2008	rev 1.2
	initialized constants with 0 for compatibility reasons
*)

END_FUNCTION

// POUs/Engineering/conversion/SPEED
FUNCTION_BLOCK SPEED
VAR_INPUT
	ms : REAL;
	kmh : REAL;
	kn : REAL;
	mh : REAL;
END_VAR
VAR_OUTPUT
	Yms : REAL;
	Ykmh : REAL;
	Ykn : REAL;
	Ymh : REAL;
END_VAR


(*
version 1.1	11. mar. 2009
programmer 	hugo
tested by		oscat

this function converts different speed units
any unused input can simply be left open.
different inputs connected at the same time will be added up.

*)

Yms := ms +
		kmh * 0.27777777777778 +
		kn * 0.5144444 +
		mh * 0.44704;
Ykmh := Yms * 3.6;
Ykn := Yms * 1.94384466037535;
Ymh := Yms * 2.23693629205440;

(*
Geschwindigkeit Meter durch Sekunde m/s 1 m/s = 3,6 km/h
km durch (pro) Stunde, nicht Stundenkilometer verwenden
Knoten kn 1 kn = 1 sm/h = 0,5144 m/s

*)

(* revision history
hm	27. mar. 2009	rev 1.0
	original version

hm	11. mar. 2009	rev 1.1
	improved code

*)

END_FUNCTION_BLOCK

// POUs/Engineering/measurements/METER
FUNCTION_BLOCK METER
VAR_INPUT
	M1, M2 : REAL;
	I1, I2 : BOOL;
	D : REAL := 1.0;
	RST : BOOL;
END_VAR
VAR_IN_OUT
	MX : REAL;
END_VAR
VAR
	MR : REAL2;
	MX1, MX2 : REAL; (* current consumption value on M1 and M2 *)
	tx: DWORD;
	last: DWORD;
	tc: REAL;
	init: BOOL;
END_VAR

(*
	version 1.4	8. mar. 2009
	programmer 	oscat
	tested BY	oscat

METER measures usage of power or similar values the output MX is the sum of the inputs over time.
MX := sum over time of (I1 * P1 + I2 * P2)/D.
a simple example is the consumption counter for a 2 stage oil burner where stage 1 is 10KW and stage 2 is 20KW.
I1 and I2 decide which value is accounted for, I1 = True only counts P1, I2 is True counts P2 
and I1 and I2 is true counts P1 and P2.
the meter can be used for all kind of consumption meters. P1 and P2 can change on the fly.

*)

(* measure the last cycle time and make sure we onle execute once every millisecond *)
tx := T_PLC_MS();
IF NOT init THEN
	init := TRUE;
	last := tx;
	mr.RX := mx;
	mr.R1 := 0.0;
ELSIF tx = last THEN
	RETURN;
ELSE
	tc := DWORD_TO_REAL(tx - last) * 0.001;
END_IF;
last := tx;

(* reset *)
IF rst THEN
	mr.R1 := 0.0;
	mr.RX := 0.0;
ELSE
	(* current consumption measurement *)
	IF I1 THEN MX1 := M1; ELSE MX1 := 0.0; END_IF;
	IF I2 THEN MX2 := M2; ELSE MX2 := 0.0; END_IF;
	(* add up the current values in a double real *)
	MR := R2_ADD(MR,(SEL(I1,0.0,mx1) + SEL(I2, 0.0, mx2)) / D * TC);
	(* set the current output value *)
	MX := mr.RX;
END_IF;




(* revision history

hm	16. sep.2007		rev 1.0
	original version

hm	7. feb 2008		rev 1.1
	use new version of ft_int to avoid a counting stop at high values
	deleted unnecessary limits

hm	24. mar. 2008	rev 1.2
	use data_type real2 to extend accuracy to 15 digits total
	do not use ft_int which adds unnecessary overhead

hm	8. feb. 2009	rev 1.3
	changed mx to be I/O
	make sure calculation works for cycle times < 1 ms

hm	8. mar. 2009	rev 1.4
	last was not updated
	code improvements

*)

END_FUNCTION_BLOCK

// POUs/Mathematical/Double Precision/R2_ADD
FUNCTION R2_ADD : REAL2
VAR_INPUT
	X : Real2;
	Y : REAL;
END_VAR
VAR
	temp: REAL;
END_VAR

(*
version 1.0	20. mar. 2008
programmer 	hugo
tested by	tobias

R2_add adds a real to a double real which extends the accuracy of a real to twice as many digits

*)

temp := X.RX;
R2_ADD.RX := Y + X.R1 + X.RX;
R2_ADD.R1 := temp - R2_ADD.RX + Y + X.R1;


(* revision history
hm		20.3.2008	rev 1.0
	original version

*)

END_FUNCTION

// POUs/Engineering/control/FT_INT
FUNCTION_BLOCK FT_INT
VAR_INPUT
	IN : REAL;
	K : REAL := 1;
	RUN : BOOL := TRUE;
	RST : BOOL;
	OUT_MIN : REAL := -1E37;
	OUT_MAX : REAL := 1E37;
END_VAR
VAR_OUTPUT
	OUT : REAL;
	LIM : BOOL;
END_VAR
VAR
	INTeg : INTEGRATE;
END_VAR


(*
version 2.2	10. mar. 2009
programmer 	hugo
tested by		oscat

FT_int is an integrator with input IN and factor K.
integration is only done while run = true, if run is false integration is stopped and the out remains at the last value.
if run is left unconnected, run is considered true by the function block.
the output ET will display the total integration time from last reset.
the out_min and out_max values can be set to ,imit the output value range. 
the default for K is 1.

 
*)

IF rst THEN
	out := 0.0;
ELSE
	integ(X := IN, E := RUN, K := K, Y := out);
END_IF;

(* limit the outputs *)
IF out >= OUT_MAX THEN
	out := out_max;
	LIM := TRUE;
ELSIF out <= out_min THEN
	out := out_min;
	lim := TRUE;
ELSE
	lim := FALSE;
END_IF;


(*
hm 13.12.2006	rev 1.1
	changed to "trapezregel" which increases accuracy
	before out := out + in * time new: out := out + (in + in_last) / 2 * time

hm 15.1.2007		rev 1.2
	added default for k to be 1.

hm	15.9.2007		rev 1.3
	replaced time() with T_PLC_US for compatibility and performance reason
	increased internal accuracy to microseconds

hm 29. oct 2007		rev 1.4
	changed code so int will not be called is time difference is 0 to increase accuracy on systems
	with cycle times below 1ms

hm	2. dec 2007	 	rev 1.5
	changed code for better performance

hm	5. jan 2008		rev 1.6
	further improvements in performance

hm	8. feb 2008		rev 1.7
	deleted limits +/- 1000 now limit is the range of real
	added variables out1 and out2 to extend the resolution
	corrected an error with elapsed time
	deleted unusfull output ET

hm	13. mar 2008	rev 1.8
	changed preset value out_min to -1e37.
	stop integrator at the limits.

hm	16. mar 2008	rev 1.9
	added type conversion to avoid warning under codesys 3.0

hm	2. jun. 2008	rev 2.0
	rewritten with clear code
	limits can now be set without run

hm	3. nov. 2008	rev 2.1
	optimized code using INTEGRATE and LIMX

hm	10. mar. 2009	rev 2.2
	removed nested comments
*)

END_FUNCTION_BLOCK

// POUs/Engineering/measurements/T_PLC_US
FUNCTION T_PLC_US : DWORD
VAR CONSTANT
	debug : BOOL := 0;
	N : INT := 0;
	offset : DWORD := 0;
END_VAR
VAR
	tx : TIME;
END_VAR

(*
version 1.2	16 nov 2008
programmer 	hugo
tested by	tobias

T_PLC_US reads the internal PLC timer and return the time, it has the advantage to be able to set a debug mode 
and speed up the counter to test the plc timer overrun which occurs every 50 days respectively 25 days at siemens S7
this routine also allows to correct the behavior of s7 where the internal plc counter will not count all 32 bits.

*)

tx := TIME();
T_PLC_US := TIME_TO_DWORD(Tx)*1000;
(* hier muss die korrektur für step7 stattfinden
plctime muss den vollen wertebereich von time ausnutzen:
wenn bei step7 time -24tage bis plus 24 tage ist dann muss der timer auch beim überlauf auf -24tage springen 
und auf keinen fall auf 0 !!!!
für siemens muss ein weiterer fb im main eingebunden werden der sicherstellt das alle 32 bits durchgezählt werden.
es kann nur ein fb sein den er muss sich das oberste (32te) bit merken.
oder etwa spring s7 bei überlauf auf -24 tage????? dann wäre keine korrektur nötig.
*)
IF debug THEN
	T_PLC_US := (SHL(T_PLC_US,N) OR SHL(DWORD#1,N)-1) + OFFSET;
END_IF;

(* revision history
hm	14.9.2007	rev 1.0
	original version

hm	12. nov 2007	rev 1.1
	added temporaray variable tx because some compilers could not handle time() as an argument

hm	16. nov. 2008	rev 1.2
	initialized constants with 0 for compatibility reasons

*)

END_FUNCTION

// POUs/Engineering/control/INTEGRATE
FUNCTION_BLOCK INTEGRATE
VAR_INPUT
	E : BOOL := TRUE;
	X : REAL;
	K : REAL := 1.0;
END_VAR
VAR_IN_OUT
	Y : REAL;
END_VAR
VAR
	X_last : REAL;
	init: BOOL;
	last: DWORD;
	tx: DWORD;
END_VAR


(*
version 1.0	3. nov. 2008
programmer 	hugo
tested by	oscat

integrate is a plain integrator with I/O for out.

 
*)

(*read system time *)
tx := T_PLC_MS();

IF NOT init THEN
	init := TRUE;
	X_last := X;
ELSIF E THEN
	Y := (X + X_LAST) * 0.5E-3 * DWORD_TO_REAL(tx-last) * K + Y;
	X_last := X;
END_IF;
last := tx;



(*
hm 3. nov. 2008	rev 1.0
original version
	
*)

END_FUNCTION_BLOCK

// POUs/Building/HLK/BURNER
FUNCTION_BLOCK BURNER
VAR_INPUT
	in : BOOL;
	stage2 : BOOL;
	over_temp : BOOL;
	oil_temp : BOOL := TRUE;
	Flame : BOOL;
	rst : BOOL;
	rst_timer : BOOL;
END_VAR
VAR_INPUT CONSTANT
	pre_heat_time : TIME := t#5s;
	pre_vent_time : TIME := t#15s;
	pre_ignite_time : TIME := t#5s;
	post_ignite_time : TIME := t#25s;
	stage2_delay : TIME := t#10s;
	safety_time : TIME := t#5s;
	lockout_time : TIME := t#10s;
	multiple_ignition : BOOL := TRUE;
	KW1 : REAL;
	KW2 : REAL;
END_VAR
VAR_OUTPUT
	motor : BOOL;
	coil1 : BOOL;
	coil2 : BOOL;
	pre_heat: BOOL;
	ignite : BOOL;
	KWh : REAL;
	status : BYTE;
	fail : BOOL;
END_VAR
VAR_IN_OUT
	runtime1 : UDINT;
	runtime2 : UDINT;
	cycles : UDINT;
END_VAR
VAR
	state : BYTE;
	last : TIME;
	tx: TIME;
	last_change: TIME;
	timer1 : ONTIME;
	timer2 : ONTIME;
	oil_temp_last: BOOL;
	cycles2 : UDINT;
END_VAR

(*
version 1.5	15 sep 2007
programmer 	oscat
tested by	oscat

burner ist eine Oel-Brenner_steuerung fuer nichtmodulierende Oelbrenner
die steuerung kann ueber setup werte programmiert werden und entsprechenden brennern angepasst werden.
die vorheizzeit ist die zeit die eine oelvorwaermung aufgeheizt wird bevor der motor gestartet wird.
der eingang oil_temp gibt an ob die oil_temp erreicht wurde, er ist default auf true und kann auch offen gelassen werden.
die vorbelueftungszeit ist die zeit die der luefter laeuft bevor die oelzufuhr freigegeben wird.
die vorzuendzeit iust diejenige zeit die die zuendung vor offnen des oelventiel gestartet wird.
nachzuendzeit ist die zeit die nach entzuendung der flamme noch gezuendet wird.
die sicherheitszeit ist die zeit nach der die oelzufuhr gesperrt wird wenn keine flamme entsteht.
nach ablauf der sicherheitszeit wird ein fehler flag gesetzt und kann erst nach der sperrzeit wieder durch einen reset geloescht werden.
waehrend der sperrzeit ist keine weitere zuendung oder einschalten moeglich.
das flag mehrfachzuendung gibt an ob eine erloschene flamme in betrieb automatisch wieder gezuendet werden soll.
der flammwaechster liegt auf eingang flamme, ein uebertemperaturschutz auf dem eingang over_temp
der betriebsstundenzaehler gibt die brennerstunden in stunden als real ausgabewer an.
der ausgang motor steuert den luefter / pumpenmotor, oil_ventil schaltet das oil ventil und zuendung schaltet die zuendung ein.

if output fail > 0 an error happened and the output has an error code:
0 :	no error
1 :	pre heating time expired and oil temp input is not true
2 :	flame monitor is active during preheating time
3 :	flame monitor active during pre_ventilation_time
4 :	no ignoition during safety time
5 :	no flame during operation
9 :	overtemp input is true

*)

(* read system time *)
tx := DWORD_TO_TIME(T_PLC_MS());

(* check rst input and overtemp *)
IF rst OR over_temp OR state = 0 THEN
	IF status > 0 AND tx - last_change >= lockout_time AND rst THEN
		status := 110;
		fail := FALSE;
		state := 1;
	ELSE
		(* normaler reset *)
		motor := FALSE;
		coil1 := FALSE;
		coil2 := FALSE;
		ignite := FALSE;
		pre_heat := FALSE;
		IF over_temp THEN
			status := 9;
			fail := TRUE;
		END_IF;
		last_change := tx;
		last := tx;
		state := 1;
	END_IF;
END_IF;

(* check for timer rst and rst timer if true *)
IF rst_timer THEN
	runtime1 := 0;
	runtime2 := 0;
	cycles := 0;
	cycles2 := 0;
END_IF;

(* quit here if an error is present *)
IF (status > 0 AND status < 100) OR rst THEN RETURN; END_IF;

(* start sequence *)
CASE state OF

1:	(* in signal starts oil pre heating *)
	IF in AND flame THEN
		state := 7;
		pre_heat := FALSE;
		status := 2;
		last_change := tx;
	ELSIF in THEN
		pre_heat := TRUE;
		state := 2;
		last_change := tx;
	END_IF;

2:	(* after pre_heating time start motor *)
	IF (tx- last_change >= pre_heat_time AND oil_temp) OR (oil_temp AND NOT oil_temp_last) THEN
		motor := TRUE;
		state := 3;
		last_change := tx;
	(* pre_heat_time ist abgelaufen und oil_temp ist nicht aktiv *)
	ELSIF tx - last_change >= pre_heat_time AND NOT oil_temp THEN
		state := 7;
		pre_heat := FALSE;
		status := 1;
		last_change := tx;
	(* flame monitor cannot be active at this time *)
	ELSIF flame THEN
		state := 7;
		pre_heat := FALSE;
		status := 2;
		last_change := tx;
	END_IF;

3:	(* abwarten bis zündung eingeschaltet werden kann *)
	IF tx - last_change >= pre_vent_time - pre_ignite_time THEN
		ignite := TRUE;
		state := 4;
		last_change := tx;
	(* flame monitor cannot be active at this time *)
	ELSIF flame THEN
		state := 7;
		pre_heat := FALSE;
		motor := FALSE;
		status := 3;
		last_change := tx;
	END_IF;

4:	(* warten bis oelzufuhr geoeffnet werden darf *)
	IF tx - last_change >= pre_ignite_time THEN
		coil1 := TRUE;
		state := 5;
		last_change := tx;
	END_IF;

5:	(* warten auf flammwaechter und falls noetig abschalten *)
	IF tx - last_change >= safety_time OR flame THEN
		IF NOT flame THEN
			(* notabschaltung da flammwaechster nicht angesprochen hat *)
			state := 7;
			motor := FALSE;
			coil1 := FALSE;
			pre_heat := FALSE;
			ignite := FALSE;
			status := 4;
			last_change := tx;
		ELSE
			state := 6;
			last_change := tx;
		END_IF;
	END_IF;

6:	(* brenner läuft, flammueberwachung und nach ablauf der nachigniteszeit ignite abschalten *)
	IF NOT flame AND NOT multiple_ignition THEN
		(* notabschaltung da flammwaechster keine flamme meldet *)
		state := 7;
		motor := FALSE;
		coil1 := FALSE;
		coil2 := FALSE;
		pre_heat := FALSE;
		ignite := FALSE;
		status := 5;
		last_change := tx;
	ELSIF NOT flame AND multiple_ignition THEN
		ignite := TRUE;
		state := 5;
		coil2 := FALSE;
		last_change := tx;
	ELSE
		IF tx - last_change >= post_ignite_time THEN
			(* post_ignite_time abgelaufen, ignite abschalten *)
			ignite := FALSE;
		END_IF;
		IF tx - last_change >= stage2_delay AND stage2 THEN
			coil2 := TRUE;
		ELSE
			coil2 := FALSE;
		END_IF;
	END_IF;
END_CASE;

(* abschaltung wenn kein eingangssignal *)
IF NOT in THEN
	state := 1;
	motor := FALSE;
	coil1 := FALSE;
	coil2 := FALSE;
	ignite := FALSE;
	pre_heat := FALSE;
	last_change := tx;
END_IF;

(* runtimezähler *)
timer1(in := flame AND in AND motor AND coil1 AND NOT coil2, seconds := runtime1, cycles := cycles);
timer2(in := flame AND in AND motor AND coil1 AND coil2, seconds := runtime2, cycles := cycles2);
KWH := UDINT_TO_REAL(runtime1) * KW1 / 3600.0 + UDINT_TO_REAL(runtime2) * KW2 / 3600.0;

(* zeit fuer naechsten aufruf merken *)
last := tx;

(* set fail output IF ERROR and Status  if normal operation *)

IF status > 0 AND status < 100 THEN
	fail := TRUE;
ELSE
	fail := FALSE;
	IF NOT in THEN
		status := 110;
	ELSIF flame AND in AND motor AND coil2 AND coil1 THEN
		status := 113;
	ELSIF flame AND in AND motor AND coil1 THEN
		status := 112;
	ELSE
		status := 111;
	END_IF;
END_IF;



(*
31.12.2006	hm		rev 1.1
	added pre_heat timing and output
	flame monitor before ignition will generate error on status output
	added output for KWh

31.12.2006	hm		rev 1.2
	added oil_temp_input

31.12.2006	hm		rev 1.3
	changed status output to be byte instead of bool

22.1.2007		hm		rev 1.4
	renamed fail output to status
	added output cycles
	corrected an error while pre_heat would be on when an error was present
	added coil2 output and stage2 input

15.9.2007		hm		rev 1.5
	replaced Time() with T_PLC_MS for compatibility and performance reasons

hm	21. oct. 2008	rev 1.6
	changed code to use new ontime rev 2.0	
*)

END_FUNCTION_BLOCK

// POUs/Engineering/measurements/ONTIME
FUNCTION_BLOCK ONTIME
VAR_INPUT
	IN : BOOL;
	RST : BOOL;
END_VAR
VAR_IN_OUT
	SECONDS : UDINT;
	CYCLES : UDINT;
END_VAR
VAR
	tx: DWORD;
	last : DWORD;
	edge : BOOL;
	init: BOOL;
	ms: DWORD;
END_VAR

(*
version 2.3	17. dec. 2008
programmer 	oscat
tested by	tobias

ONTIME measures the ontime of a signal in seconds.
the output SECONDS is of type DWORD which results in a total measurement range of 1 second up to 136 years.
internally ontime works with a resolution of milliseconds

*)

(* read system time *)
tx := T_PLC_MS();

(* make sure the first cycle works correctly *)
IF NOT init OR rst THEN
	init := TRUE;
	last := tx;
	SECONDS := 0;
	CYCLES := BOOL_TO_UINT(in);
	ms := 0;
ELSIF IN THEN
	(* add the current milliseconds *)
	ms := (tx - last) + ms;
	IF ms >= 1000 THEN
		seconds := seconds + 1;
		ms := ms - 1000;
	END_IF;
	cycles := cycles + BOOL_TO_UINT(NOT edge);
END_IF;
last := tx;
edge := in;


(* revision history
hm 22.2.2007		rev 1.1
	changed VAR RETAIN PERSISTENT to VAR RETAIN for better compatibility
	wago lon contollers do not support persisitent

hm 2.8.2007		rev 1.2
	adding time up in a real number will automatically lead to the point where 
	small time scales like the cycle time will be below the resolution of real and therefore
	ontime would not increase in small steps as necessary
	the time is now measured internally in two  dwords and be converted to real only for
	output purposes.
	deleted the variable power because it was unnecessary

hm	16.9.2007		rev 1.3
	changes time() to T_plc_ms() for compatibility reasons

hm	2. dec. 2007	rev 1.4
	chaged code for better performance

hm	16. mar. 2008	rev 1.5
	added type conversions to avoid warnings under codesys 3.0

hm	21. oct. 2008	rev 2.0
	changed module for much better performance and allow for external result storage

hm	10. nov. 2008	rev 2.1
	increased internal resolution to milliseconds

hm	16. nov. 2008	rev 2.2
	changed typecast to avoid warnings

hm	17. dec. 2008	rev 2.3
	fixed an error when in would be true for more then 49 days
*)

END_FUNCTION_BLOCK

// POUs/Time&Date/SECOND
FUNCTION SECOND : REAL
VAR_INPUT
	itod : TOD;
END_VAR


(*
version 1.1	2 oct 2006
programmer 	hugo
tested by	oscat

returns the seconds and milliseconds as real of TOD   
 
*)

SECOND := DWORD_TO_REAL(TOD_TO_DWORD(itod) - TOD_TO_DWORD(itod)/60000 * 60000) / 1000;



(* change history

hm	2. oct. 2006 rev 1.1 
	changed name of input to itod

*)

END_FUNCTION

// POUs/Mathematical/Array/_ARRAY_INIT
FUNCTION _ARRAY_INIT : BOOL
VAR_INPUT
	pt : POINTER TO ARRAY[0..32000] OF REAL;
	size : UINT;
	init : REAL;
END_VAR
VAR
	i: UINT;
	stop: UINT;
END_VAR


(*
version 1.3	16 mar 2008
programmer 	hugo
tested by		tobias

this function will initialize a given array with a value init.
the function needs to be called:	_array_init(adr("array"),sizeof("array"));
this function will manipulate a given array.
the function manipulates the original array, it rerturnes true when finished.
because this function works with pointers its very time efficient and it needs no extra memory.

*)

stop := SHR(size,2)-1;
FOR i := 0 TO stop DO
	pt^[i] := init;
END_FOR;

_array_init := TRUE;

(* revision History

hm 6.1.2007		rev 1.1
	change type of function to bool
	added  array_init := true to set output true.

hm	14.11.2007	rev 1.2
	changed stop calculation to be more efficient

hm	16.3. 2008		rev 1.3
	changed type of input size to uint
*)

END_FUNCTION

// POUs/Mathematical/Array/_ARRAY_MEDIAN
FUNCTION _ARRAY_MEDIAN : REAL
VAR_INPUT
	pt : POINTER TO ARRAY[0..32000] OF REAL;
	size : UINT;
END_VAR
VAR
	i: UINT;
	stop: UINT;
END_VAR

(*
version 1.5	16 mar 2008
programmer 	hugo
tested by		tobias

this function will calculate the median of a given array.
in order to do so the ariginal array is sorted and stays sorted after the function finishes
the function needs to be called:	_array_median(adr("array"),sizeof("array"));
this function will manipulate a given array.
the function will return the median of the original array.
for example [12,0,4,7,1] the median is 4 and the array after the function is called is [0,1,4,7,12]
because this function works with pointers its very time efficient and it needs no extra memory.

*)

_ARRAY_SORT(pt,size);
stop := SHR(size,2)-1;
IF EVEN(UINT_TO_INT(stop)) THEN
	_ARRAY_MEDIAN := pt^[SHR(stop,1)];
ELSE
	i := SHR(stop,1);
	_ARRAY_MEDIAN := (pt^[i] + pt^[i+1]) * 0.5;
END_IF;

(* old code
stop := (size - SIZEOF(pt)) / SIZEOF(pt);
FOR i := 0 TO stop - 1 DO
	FOR m := i + 1 TO stop DO
		IF pt^[i] > pt^[m] THEN
			temp := pt^[i];
			pt^[i] := pt^[m];
			pt^[m] := temp;
		END_IF;
	END_FOR;
END_FOR;
IF even(stop) THEN
	_array_median := pt^[stop/2];
ELSE
	i := stop/2;
	_array_median := (pt^[i] + pt^[i+1])/2;
END_IF;
*)
(* revision history
hm 	3.3.2007		rev 1.1
	corrected an error, changed the statement line 14	i := TRUNC(stop/2); to i := stop/2;

hm		22. sep 2007	rev 1.2
	changed algorithm to use _array_soft for performance reasons

hm		8. oct 2007		rev 1.3
	deleted unused variables m and temp

hm		14. nov 2007	rev 1.4
	corrected a problem with size calculation

hm		16.3. 2008		rev 1.5
	changed type of input size to uint
	performance improvements
*)

END_FUNCTION

// POUs/Mathematical/Array/_ARRAY_SORT
FUNCTION _ARRAY_SORT : BOOL
VAR_INPUT
	pt : POINTER TO ARRAY[1..32000] OF REAL;
	size : UINT;
END_VAR
VAR
	i: INT;
	j: INT;
	temp : REAL;
	stop : INT;
	heapsize: INT;
	popmax : REAL;
	size2: INT;
	hs2: INT;
END_VAR

(*
version 1.6	16. mar. 2008
programmer 	hugo
tested by		tobias

this function will sort a given array.
the function needs to be called:	_array_sort(adr("array"),sizeof("array"));
this function will manipulate a given array.
the function will not return anything except true, it will instead manipulate the original array.
because this function works with pointers its very time efficient and it needs no extra memory.

*)

(* generate heap *)

size := SHR(size,2);
size2 := UINT_TO_INT(SHR(size,1));
FOR i := SIZE2  TO 1 BY -1 DO 		(* zweite Hälfte des Feldes braucht nicht betrachtet werden *)
	j:=i;
    WHILE j <= SIZE2 DO
     	stop := j * 2 + 1;               (* finde Maximum der (beiden) Söhne *)
        IF stop > UINT_TO_INT(SIZE) THEN stop := stop - 1;
        ELSIF pt^[stop-1] > pt^[stop] THEN stop := stop - 1;
		END_IF;
        IF pt^[j] < pt^[stop] THEN   		(* ggf. tauschen *)
         	temp := pt^[j];
            pt^[j] := pt^[stop];
            pt^[stop] := temp;
        END_IF;
        j := stop;
    END_WHILE;
END_FOR;

(* heapsort *)
FOR heapsize := UINT_TO_INT(size) TO 1 BY -1 DO
	popmax := pt^[1];
	pt^[1] := pt^[heapsize];
   	i := 1;
	hs2 := SHR(heapsize,1);
	WHILE i <= hs2 DO	     (* letztes Element an Anfang setzen und versickern lassen *)
       	stop := i * 2 + 1;                (* finde Maximum der (beiden) Söhne *)
        	IF stop > heapsize THEN stop := stop - 1;
        	ELSIF pt^[stop-1] > pt^[stop] THEN stop := stop - 1;
	 	END_IF;
        	IF pt^[i] < pt^[stop] THEN	     (* ggf. tauschen *)
            		temp := pt^[i];
            		pt^[i] := pt^[stop];
            		pt^[stop] := temp;
        	END_IF;
        	i := stop;
    	END_WHILE;
	pt^[heapsize] := popmax;
END_FOR;

_ARRAY_SORT := TRUE;

(* old algorithm bubble sort used before rev 1.2
stop := (size - SIZEOF(pt)) / SIZEOF(pt);
FOR i := 0 TO stop - 1 DO
	FOR m := i + 1 TO stop DO
		IF pt^[i] > pt^[m] THEN
			temp := pt^[i];
			pt^[i] := pt^[m];
			pt^[m] := temp;
		END_IF;
	END_FOR;
END_FOR;
_array_sort := TRUE;

*)
(* revision history

hm 	6.1.2007 	rev 1.1
	changed return value to true

hm	22. sep 2007	rev 1.2
	changed sorting algorithm to heap sort for performance reasons

hm 	14. nov 2007	rev 1.3
	changed calculation of stop to be more efficient

hm	15 dec 2007	rev 1.4
	added function return true

hm	5. jan 2008		rev 1.5
	improved performance

hm	16. mar. 2008	rev 1.6
	changed type of input size to uint

hm	28. mar. 2008	rev 1.7
	changed input f to pt

*)

END_FUNCTION

// POUs/Mathematical/EVEN
FUNCTION EVEN : BOOL
VAR_INPUT
	in : DINT;
END_VAR


(*
version 1.1	1 dec 2007
programmer 	hugo
tested by		tobias

this function chacks an input for even  value
the output is true if the input is even.
execution time on wago 750 - 841 =  10  us
*)

EVEN := NOT in.0;

(* revision history
hm	1. oct 2006	rev 1.0
	ORIGINAL VERSION

hm	01.12.2007	rev 1.1
	changed code for improved performance

hm	21. mar. 2008	rev 1.2
	changed type of input IN from INT to DINT
*)

END_FUNCTION

// POUs/Mathematical/Array/_ARRAY_MUL
FUNCTION _ARRAY_MUL : BOOL
VAR_INPUT
	pt : POINTER TO ARRAY[0..32000] OF REAL;
	size : UINT;
	X : REAL;
END_VAR
VAR
	i: UINT;
	stop: UINT;
END_VAR

(*
version 1.0	2. apr. 2008
programmer 	hugo
tested by	tobias

this function will multiply each element of the array and stroe the result instead of the element.
Array[i] := ARRAY[i] * X.
the function needs to be called:	array_avg(adr("array"),sizeof("array"));
because this function works with pointers its very time efficient and it needs no extra memory.

*)

stop := SHR(size,2)-1;
FOR i := 0 TO stop DO
	PT^[i] := PT^[i] * X;
END_FOR;
_ARRAY_MUL := TRUE;


(* revision history
hm	2. apr 2008		rev 1.0
	original version

*)

END_FUNCTION

// POUs/Mathematical/Array/_ARRAY_SHUFFLE
FUNCTION _ARRAY_SHUFFLE : BOOL
VAR_INPUT
	pt : POINTER TO ARRAY[0..32000] OF REAL;
	size : UINT;
END_VAR
VAR
	temp : REAL;
	pos  : INT;
	i: INT;
	stop: INT;
END_VAR


(*
version 1.2	30. mar. 2008
programmer 	kurt
tested by		hugo

this function will randomly shuffle the elements of an array
*)

stop := UINT_TO_INT(SHR(size,2)-1);
FOR i := 0 TO stop DO
        pos := RDM2(i+pos,0,stop);
        (* swap elements *)
        temp := pt^[i];
        pt^[i] := pt^[pos];
        pt^[pos] := temp;
END_FOR;

_ARRAY_SHUFFLE := TRUE;


(* revision History
hm 	4. mar 2008	rev 1.0
	original version

hm	16. mar. 2008	rev 1.1
	changed type of input size to uint

hm	30. mar. 2008	rev 1.2
	changed last in rdm2 fromm pos to i + pos to allow for more randomness

*)

END_FUNCTION

// POUs/Mathematical/RDM2
FUNCTION RDM2 : INT
VAR_INPUT
	last : INT;
	low : INT;
	high : INT;
END_VAR


(*
version 1.1	18. oct. 2008
programmer 	hugo
tested by	tobias

this function calculates an integer pseudo random number
the random number will be in the range of low <= rdm2 <= high.

*)

RDM2 := TRUNC_INT(RDM(FRACT(last * math.PI)) * (high - low + 1)) + low;

(* revision history
hm		29. feb 2008		rev 1.0
	original version

hm		18. oct. 2008		rev 1.1
	using math constants

*)

END_FUNCTION

// POUs/Mathematical/RDM
FUNCTION RDM : REAL
VAR_INPUT
	last : REAL;
END_VAR
VAR
	tn : DWORD;
	tc : INT;
END_VAR


(*
version 1.9	10. mar. 2009
programmer 	hugo
tested by		tobias

this function calculates a pseudo random number
to generate the number it reads the sps timer and calculates a random number between 0 and 1:
in order to use rdm more then once within one sps cycle it need to be called with different seed numbers LAST.

*)

tn := T_PLC_MS();
tc := BIT_COUNT(tn);
tn.31 := tn.2;
tn.30 := tn.5;
tn.29 := tn.4;
tn.28 := tn.1;
tn.27 := tn.0;
tn.26 := tn.7;
tn.25 := tn.6;
tn.24 := tn.3;
tn := ROL(tn,BIT_COUNT(tn)) OR 16#80000001;
tn := tn MOD 71474513 + INT_TO_DWORD(tc + 77);
RDM := FRACT(DWORD_TO_REAL(tn) / 10000000.0 * (math.E - LIMIT(0.0,last,1.0)));


(*
pt := ADR(temp);
pt^ := (T_PLC_MS() AND 16#007FFFFF) OR 16#3D000000;
RDM := fract(modR(temp*e+pi1, PI1-last) + modR(temp*PI1+e + last,e-last));
*)

(* revision history
hm		16. jan 2007		rev 1.0
	original version

hm		11. nov 2007		rev 1.1
	changed time() into t_plc_ms()

hm		20. nov 2007		rev 1.2
	changed code of temp calculation to avoid overflow in modr due to resuclt would not fit DINT for high timeer values

hm		5. jan 2008		rev 1.3
	changed calculation of temp to avoid problem with high values of t_plc_ms

hm		2. feb 2008		rev 1.4
	changed algorithm to avoind non iec functions and guarantee more randomness

hm	10. mar. 2008		rev 1.5
	make sure last will be between 0 and 1 to avoid invalid results

hm	16. mar. 2008		rev 1.6
	added conversion for tc to avoid warnings under codesys 3.0

hm	18. may. 2008		rev 1.7
	changed constant E to E1

hm	18. oct. 2008		rev 1.8
	using math constants

hm	10. mar. 2009		rev 1.9
	real constants updated to new systax using dot

*)

END_FUNCTION

// POUs/Logic/gate logic/BIT_COUNT
FUNCTION BIT_COUNT : INT
VAR_INPUT
	IN : DWORD;
END_VAR


(*
version 1.1	10 sep 2007
programmer 	hugo
tested by		tobias

BIT_COUNT counts the amount True of bits in a dword.
for exabple: bit_count(3) returns 2 because two bits (bits 0 and 1) are true and all others are false. 

*)

WHILE in > 0 DO
	IF in.0 THEN Bit_Count := Bit_Count + 1; END_IF;
	in := SHR(in,1);
END_WHILE;



(* revision history
5.7.2007	rev 1.0		original version

10.9.2007	rev 1.1		hm
	changed algorithm for better performace
	the execution time has reduced by a factor of 5
	deleted unused variable temp
*)

END_FUNCTION

// POUs/Mathematical/FRACT
FUNCTION FRACT : REAL
VAR_INPUT
	x : REAL;
END_VAR


(*
version 1.3	10. mar. 2009
programmer 	hugo
tested by		tobias

this function returns the fraction of a real number
fract(3.14) = 0.14

*)

IF ABS(x) < 2.0E9 THEN
	FRACT := x - DINT_TO_REAL(D_TRUNC(x));
ELSE
	FRACT := 0.0;
END_IF;

(* revision history
hm	4. aug 2006	rev 1.0
	original version

hm	11. mar 2008	rev 1.1
	added dint_to_real for compatibility reasons
	now returns 0 for number > 2e9
	changed input to x

hm	21. mar. 2008	rev 1.2
	use D_trunc instead of TRUNC for compatibility reasons

hm	10. mar. 2009	rev 1.3
	real constants updated to new systax using dot

*)

END_FUNCTION

// POUs/Mathematical/D_TRUNC
FUNCTION D_TRUNC : DINT
VAR_INPUT
	X : REAL;
END_VAR

(*
version 1.2	10. mar. 2009
programmer 	hugo
tested by		oscat

d_trunc truncates a real to a dint 1.5 will be 1 and -1.5 will be -1
d_trunc is necessary because many systems do not offer a trunc to a dint
also real_to_dint will not deliver the same result on different systems

*)

D_TRUNC := REAL_TO_DINT(X);
IF X > 0.0 THEN
	IF DINT_TO_REAL(D_TRUNC) > X THEN D_TRUNC := D_TRUNC - 1; END_IF;
ELSE
	IF DINT_TO_REAL(D_TRUNC) < X THEN D_TRUNC := D_TRUNC + 1; END_IF;
END_IF;


(* for systems that support a dint truncation this routine can be replaced by trunc() *)


(* revision history
hm	21. mar. 2008	rev 1.0
	original version

hm	31. oct. 2008	rev 1.1
	optimized performance

hm	10. mar. 2009	rev 1.2
	real constants updated to new systax using dot
*)

END_FUNCTION

// POUs/Mathematical/MODR
FUNCTION MODR : REAL
VAR_INPUT
	IN : REAL;
	DIVI : REAL;
END_VAR


(*
version 1.5	10. mar. 2009
programmer 	hugo
tested by		tobias

this is a modulo funtion for real numbers
modr(5.5,2.5) = 0.5

*)

IF divi = 0.0 THEN
	MODR := 0.0;
ELSE
	MODR := in - DINT_TO_REAL(FLOOR2(in / divi)) * divi;
END_IF;

(* revision history

hm	4. aug.2006		rev 1.0

hm	28. jan.2007	rev 1.1
	modr(x,0) will deliver the result 0

hm	21. mar 2008	rev 1.2
	use D_trunc for compatibility reasons

hm	4. apr. 2008	rev 1.3
	added type conversion to avoid warnings under codesys 3.0

hm	31. oct. 2008	rev 1.4
	changed algorithm to the more common version using floor instead of TRUNC

hm	10. mar. 2009	rev 1.5
	real constants updated to new systax using dot

*)

END_FUNCTION

// POUs/Mathematical/FLOOR2
FUNCTION FLOOR2 : DINT
VAR_INPUT
	X : REAL;
END_VAR



(*
version 1.1	4. apr. 2008
programmer 	hugo
tested by		tobias

This is a rounding function which returns the biggest possible integer which is less or equal to X.
floor2(3.14) = 3
floor2(-3.14) = -4

*)

FLOOR2 := REAL_TO_DINT(X);
IF DINT_TO_REAL(FLOOR2) > X THEN
	FLOOR2 := FLOOR2 - 1;
END_IF;

(* revision history
hm	21. mar. 2008	rev 1.0
	originlal version

hm	4. apr. 2008	rev 1.1
	added type conversion to avoid warnings under codesys 3.0
*)

END_FUNCTION

// POUs/Mathematical/FLOOR
FUNCTION FLOOR : INT
VAR_INPUT
	X : REAL;
END_VAR


(*
version 1.1	21. mar. 2008
programmer 	hugo
tested by		tobias

This is a rounding function which returns the biggest possible integer which is less or equal to X.
floor(3.14) = 3
floor(-3.14) = -4

*)

FLOOR := REAL_TO_INT(X);
IF FLOOR > X THEN
	FLOOR := FLOOR - 1;
END_IF;

(* revision history
hm		7. feb 2007		rev 1.0
	originlal version

hm		21. mar. 2008	rev 1.1
	replaced trunc with real_to_int for compatibility reasons

*)

END_FUNCTION

// POUs/Buffer Management/_BUFFER_CLEAR
FUNCTION _BUFFER_CLEAR : BOOL
VAR_INPUT
	PT : POINTER TO BYTE;
	SIZE : UINT;
END_VAR
VAR
	ptw : POINTER TO DWORD;
	temp: DWORD;
	end, end32 : DWORD;
END_VAR


(*
version 1.2	31. oct. 2008
programmer 	hugo
tested by	oscat

this function will initialize a given array of byte with 0.
the function needs to be called:	_buffer_clear(adr("array"),sizeof("array"));
this function will manipulate a given array.
the function manipulates the original array, it rerturnes true when finished.
because this function works with pointers its very time efficient and it needs no extra memory.

*)

(* this routine uses 32 bit access to gain speed *)
(* first access bytes till pointer is aligned for 32 bit access *)
temp := pt;
end := temp + UINT_TO_DWORD(size);
end32 := end - 3;
WHILE (pt < end) AND ((temp AND 16#00000003) > 0) DO
	pt^ := 0;
	pt := pt + 1;
	temp := temp + 1;
END_WHILE;
(* pointer is aligned, now copy 32 bits at a time *)
ptw := pt;
WHILE ptw < end32 DO (* *)
	ptw^ := 0;
	ptw := ptw + 4;
END_WHILE;
(* copy the remaining bytes in byte mode *)
pt := ptw;
WHILE pt < end DO
	pt^ := 0;
	pt := pt + 1;
END_WHILE;

_BUFFER_CLEAR := TRUE;

(* revision History
hm 	5. mar. 2008	rev 1.0
	original version

hm	16. mar. 2008	rev 1.1
	added type conversion to avoid warnings under codesys 30
	chaged type of input size to uint
	deleted unused variable i

hm	31. oct. 2008	rev 1.2
	corrected an error while routine would write outside of arrays

*)

END_FUNCTION

// POUs/Buffer Management/_BUFFER_INIT
FUNCTION _BUFFER_INIT : BOOL
VAR_INPUT
	PT : POINTER TO BYTE;
	SIZE : UINT;
	INIT : BYTE;
END_VAR
VAR
	ptw : POINTER TO DWORD;
	temp : DWORD;
	end, end32 : DWORD;
END_VAR


(*
version 1.2	31. oct. 2008
programmer 	hugo
tested by	oscat

this function will initialize a given array of byte with init.
the function needs to be called:	_buffer_init(adr("array"),sizeof("array"),init);
this function will manipulate a given array.
the function manipulates the original array, it rerturnes true when finished.
because this function works with pointers its very time efficient and it needs no extra memory.

*)

(* this routine uses 32 bit access to gain speed *)
(* first access bytes till pointer is aligned for 32 bit access *)
temp := pt;
end := temp + UINT_TO_DWORD(size);
end32 := end - 3;
WHILE (pt < end) AND ((temp AND 16#00000003) > 0) DO
	pt^ := init;
	pt := pt + 1;
	temp := temp + 1;
END_WHILE;
(* pointer is aligned, now copy 32 bits at a time *)
ptw := pt;
temp := SHL(BYTE_TO_DWORD(init),24) OR SHL(BYTE_TO_DWORD(init),16) OR SHL(BYTE_TO_DWORD(init),8) OR BYTE_TO_DWORD(init);
WHILE ptw < end32 DO
	ptw^ := temp;
	ptw := ptw + 4;
END_WHILE;
(* copy the remaining bytes in byte mode *)
pt := ptw;
WHILE pt < end DO
	pt^ := init;
	pt := pt + 1;
END_WHILE;

_BUFFER_INIT := TRUE;

(* revision History
hm 	5. mar. 2008	rev 1.0
	original version

hm	16. mar. 2008	rev 1.1
	added type conversion to avoid warnings under codesys 3.0
	chaged type of input size to uint.

hm	31. oct. 2008	rev 1.2
	corrected an error while routine would write outside of arrays

*)

END_FUNCTION

// POUs/Buffer Management/_BUFFER_INSERT
FUNCTION _BUFFER_INSERT : BOOL
VAR_INPUT
	STR : STRING(STRING_LENGTH);
	POS : INT;
	PT : POINTER TO ARRAY[0..32767] OF BYTE;
	SIZE : UINT;
END_VAR
VAR
	end : INT;
	lx: INT;
	i: INT;
END_VAR


(*
version 1.4	12. nov. 2009
programmer 	hugo
tested by		oscat

this function will initialize a given array of byte with init.
the function needs to be called:	_buffer_init(adr("array"),sizeof("array"),init);
this function will manipulate a given array.
the function manipulates the original array, it rerturnes true when finished.
because this function works with pointers its very time efficient and it needs no extra memory.

*)

lx := LEN(str);
end := pos + lx;
(* first move the upper part of the buffer to make space for the string *)
FOR i := UINT_TO_INT(size) - 1 TO end BY -1 DO
	pt^[i] := pt^[i-lx];
END_FOR;
(* copy the string *)
_BUFFER_INSERT := _STRING_TO_BUFFER(str, pos, PT, size);


(* revision History
hm 	9. mar. 2008	rev 1.0
	original version

hm	16. mar. 2008	rev 1.1
	changed type of input size to uint

hm	13. may. 2008	rev 1.2
	changed type of pointer to array[1..32767]
	changed size of string to STRING_LENGTH

hm	23. mar. 2009	rev 1.3
	avoid writing to input pos

hm	12. nov. 2009	rev 1.4
	code optimized

*)

END_FUNCTION

// POUs/Buffer Management/_STRING_TO_BUFFER
FUNCTION _STRING_TO_BUFFER : BOOL
VAR_INPUT
	STR : STRING(STRING_LENGTH);
	POS : INT;
	PT : POINTER TO ARRAY[0..32767] OF BYTE;
	SIZE : UINT;
END_VAR
VAR
	ps : POINTER TO BYTE;
	i: INT;
	end: INT;
END_VAR


(*
version 1.3	12. nov. 2009
programmer 	hugo
tested by		oscat

this function will copy a string into an array of byte starting at position pos.
the function needs to be called:	_String_To_buffer(str, pos, adr("array"),sizeof("array"));
this function will manipulate the array directly in memory and returns true when finished.
because this function works with pointers its very time efficient and it needs no extra memory.

*)

ps := ADR(str);
end := MIN(pos + LEN(str), UINT_TO_INT(size));
IF end > 0 THEN end := end -1; END_IF;
FOR i := pos TO end DO
	pt^[i] := ps^;
	ps := ps + 1;
END_FOR;

_STRING_TO_BUFFER := TRUE;

(* revision History

hm 	5. mar. 2008	rev 1.0
	original version

hm	16. mar. 2008	rev 1.1
	changed type of input size to uint

hm	13. may. 2008	rev 1.2
	changed type of pointer to array[1..32767]
	changed size of string to STRING_LENGTH

hm	12. nov. 2009	rev 1.3
	limit end to size - 1

*)

END_FUNCTION

// POUs/Engineering/signal generators/_RMP_B
FUNCTION_BLOCK _RMP_B
VAR_INPUT
	DIR : BOOL;  (* true = up *)
	E : BOOL := TRUE;
	TR : TIME;
END_VAR
VAR_IN_OUT
	RMP : BYTE;
END_VAR
VAR
	tx, tl : DWORD;
	step : INT;
	init: BOOL;
	last_dir: BOOL;
END_VAR


(*
version 1.1	20. nov. 2008
programmer 	hugo
tested by	oscat


_RMP_B generates a ramp on an external var of type byte
tr is the total ramp time, E is an enable and dir the direction of the ramp

*)

tx := T_PLC_MS();
IF E AND init THEN
	(* we need to set tl = tx when direction changes *)
	IF dir XOR last_dir THEN
	 tl := tx;
	 last_dir := dir;
	END_IF;
	(* check_elapsed time and calculate only if necessary *)
	IF tr > t#0s THEN
		step := DWORD_TO_INT(SHL(tx-tl, 8) / TIME_TO_DWORD(TR));
	ELSE
		step := 255;
	END_IF;
	IF step > 0 THEN
		(* perform the step on the ramp *)
		tl := tx;
		(* calculate the step response *)
		IF NOT dir THEN step := - step; END_IF;
		rmp := INT_TO_BYTE(LIMIT(0, BYTE_TO_INT(rmp) + step, 255));
	END_IF;
ELSE
	tl := tx;
	init := TRUE;
END_IF;


(* revison history
hm	22. oct. 2008	rev 1.0
	original version

hm	20. nov. 2008	rev 1.1
	set default for E to be TRUE
	added init

*)

END_FUNCTION_BLOCK

// POUs/Engineering/signal generators/_RMP_NEXT
FUNCTION_BLOCK _RMP_NEXT
VAR_INPUT
	E : BOOL := TRUE;
	IN : BYTE;
	TR : TIME;
	TF : TIME;
	TL : TIME;
END_VAR
VAR_OUTPUT
	DIR : BOOL;    (* upwards = TRUE *)
	UP : BOOL;
	DN : BOOL;
END_VAR
VAR_IN_OUT
	OUT : BYTE;
END_VAR
VAR
	rmx : _RMP_B;
	dirx : TREND_DW;
	t_lock :TP;
	xen: BOOL;
	xdir: BOOL;
END_VAR


(*
version 1.4	18. jul. 2009
programmer 	hugo
tested by		oscat


_RMP_NEXT  will generate a ramp output following the input IN.
on a rising ramp the output will stop as soon as it has surpassed the input in, and on a falling ramp it will stop when out is smaller than in.
a lockout time T_L will be added between up and down direction.

*)

dirx(X := in);

t_lock(in := FALSE, pt := TL);

IF dirx.TU AND (OUT < IN) THEN
	IF NOT xdir AND xen THEN t_lock(in := TRUE); END_IF;
	xen := TRUE;
	xdir := TRUE;
ELSIF dirx.TD AND (OUT > IN) THEN
	IF xdir AND xen THEN t_lock(in := TRUE); END_IF;
	xen := TRUE;
	xdir := FALSE;
ELSIF xen THEN
	IF (xdir AND (out >= in)) OR (NOT xdir AND (out <= in)) THEN
		xen := FALSE;
		IF tl > t#0s THEN t_lock(IN := TRUE); END_IF;
	END_IF;
END_IF;

IF NOT t_lock.Q AND xen THEN
		UP := XDIR;
		DIR := XDIR;
		DN := NOT XDIR;
ELSE
	UP := FALSE;
	DN := FALSE;
END_IF;

rmx(rmp := OUT, E := E AND (UP OR DN) , dir := DIR, tr := SEL(dir, TF, TR));


(* revison history
hm	23. nov. 2008	rev 1.0
	original version

hm	24. jan. 2009	rev 1.1
	deleted unused vars tmp1, tmp2

hm	20. feb. 2009	rev 1.2
	improved algorithm
	added TL

hm	9. mar. 2009	rev 1.3
	input E was ignored
	removed double assignments

hm	18. jul. 2009	rev 1.4
	improved performance

*)

END_FUNCTION_BLOCK

// POUs/Engineering/signal processing/TREND_DW
FUNCTION_BLOCK TREND_DW
VAR_INPUT
	X : DWORD;
END_VAR
VAR_OUTPUT
	Q : BOOL;
	TU : BOOL;
	TD : BOOL;
	D : DWORD;
END_VAR
VAR
	last_X: DWORD;
END_VAR

(*
version 1.2	14. mar. 2009
programmer 	hugo
tested by		oscat

trend_DW analyses the trend of a input signal.
The Output Q is True if the input X is >= last_X and is false if the input X is <= last_X
in addition to the trend the output TU will be high for one cycle to signal a rising of the input value X
and  TD will signal a decreasing value on the input X.
in case of a change the output D will show the delta of the input to the last input value.


*)

IF X > last_X THEN
	TU := TRUE;
	TD := FALSE;
	D := X - last_X;
	Q := TRUE;
ELSIF X < last_X THEN
	TD := TRUE;
	TU := FALSE;
	D := last_X - X;
	Q := FALSE;
ELSE
	TU := FALSE;
	TD := FALSE;
	D := 0;
END_IF;
last_X := X;



(* revision history
hm	21. nov. 2008	rev 1.0
	original version

hm	20. feb. 2009	rev 1.1
	added outputs TU, TD and D

hm	14. mar. 2009	rev 1.2
	removed double assignments

*)

END_FUNCTION_BLOCK

// POUs/Engineering/signal processing/TREND
FUNCTION_BLOCK TREND
VAR_INPUT
	X : REAL;
END_VAR
VAR_OUTPUT
	Q : BOOL;
	TU : BOOL;
	TD : BOOL;
	D : REAL;
END_VAR
VAR
	last_X: REAL;
END_VAR

(*
version 1.0	21. aug. 2009
programmer 	hugo
tested by		oscat

trend analyses the trend of a input signal.
The Output Q is True if the input X is >= last_X and is false if the input X is <= last_X
in addition to the trend the output TU will be high for one cycle to signal a rising of the input value X
and  TD will signal a decreasing value on the input X.
in case of a change the output D will show the delta of the input to the last input value.

*)

TU := X > last_X;
TD := X < last_X;
Q := TU OR TD;
D := X - LAST_X;

last_X := X;



(* revision history
hm	21. aug. 2009	rev 1.0
	original version

*)

END_FUNCTION_BLOCK

// POUs/Engineering/signal generators/_RMP_W
FUNCTION_BLOCK _RMP_W
VAR_INPUT
	DIR : BOOL;
	E : BOOL := TRUE;
	TR : TIME;
END_VAR
VAR_IN_OUT
	RMP : WORD;
END_VAR
VAR
	tx, tl : DWORD;
	step : DINT;
	init: BOOL;
	last_dir : BOOL;
END_VAR


(*
version 1.1	20. nov. 2008
programmer 	hugo
tested by	oscat


_RMP_B generates a ramp on an external var of type byte
tr is the total ramp time, E is an enable and dir the direction of the ramp

*)

tx := T_PLC_MS();
IF E AND init THEN
	(* we need to set tl = tx when direction changes *)
	IF dir XOR last_dir THEN
	 tl := tx;
	 last_dir := dir;
	END_IF;
	(* check_elapsed time and calculate only if necessary *)
	IF tr > t#0s THEN
		step := DWORD_TO_DINT(SHL(tx-tl, 16) / TIME_TO_DWORD(TR));
	ELSE
		step := 65535;
	END_IF;
	IF step > 0 THEN
		(* perform the step on the ramp *)
		tl := tx;
		(* calculate the step response *)
		IF NOT dir THEN step := - step; END_IF;
		rmp := DINT_TO_WORD(LIMIT(0, WORD_TO_DINT(rmp) + step, 65535));
	END_IF;
ELSE
	tl := tx;
	init := TRUE;
END_IF;


(* revison history
hm	22. oct. 2008	rev 1.0
	original version

hm	20. nov. 2008	rev 1.1
	set default for E to be TRUE
	added init

*)

END_FUNCTION_BLOCK

// POUs/Logic/generators/A_TRIG
FUNCTION_BLOCK A_TRIG
VAR_INPUT
	IN : REAL;
	RES : REAL;
END_VAR
VAR_OUTPUT
	Q : BOOL;
	D : REAL;
END_VAR
VAR
	last_in : REAL;
END_VAR

(*
version 1.1	25. oct. 2008
programmer 	hugo
tested by	oscat

this block is similar to the IEC Standard R_trig and F_trig but it monitors a REAL for change.
if the valiue on IN changes more then D from the last value it will generate trigger and display the difference in output D.
the trigger will only be active for one cycle.

*)

D := IN - LAST_IN;
Q := ABS(D) > res;
IF Q THEN last_in := IN; END_IF;
D := IN - LAST_IN;


(* revision history

hm 	16. jul. 2008	rev 1.0
	original version released

hm	25. oct. 2008	rev 1.1
	code optimization
	a_trig now also works for res = 0

*)

END_FUNCTION_BLOCK

// POUs/Mathematical/ACOSH
FUNCTION ACOSH : REAL
VAR_INPUT
	X : REAL;
END_VAR


(*
version 1.3	10. mar. 2009
programmer 	hugo
tested by		tobias

this function calculates the arcus cos hyperbolicus

*)

ACOSH := LN(SQRT(X * X - 1.0) + X);

(* revision history
hm		12 jan 2007	rev 1.0
	original version

hm		2. dec 2007	rev 1.1
	changed code for better performance

hm	16. mar. 2007		rev 1.2
	changed sequence of calculations to improve performance

hm	10. mar. 2009		rev 1.3
	real constants updated to new systax using dot

*)

END_FUNCTION

// POUs/Mathematical/ACOTH
FUNCTION ACOTH : REAL
VAR_INPUT
	X : REAL;
END_VAR


(*
version 1.2	10. mar. 2009
programmer 	hugo
tested by		tobias

this function calculates the arcus cotangens hyperbolicus

*)

ACOTH := LN((x+1.0)/(x-1.0))*0.5;

(* revision history
hm		12 jan 2007	rev 1.0
	original version

hm		5. jan 2008	rev 1.1
	improved code for better performance

hm	10. mar. 2009		rev 1.2
	real constants updated to new systax using dot

*)

END_FUNCTION

// POUs/Building/actuators/ACTUATOR_2P
FUNCTION_BLOCK ACTUATOR_2P
VAR_INPUT
	IN : BYTE;
	TEST : BOOL;
	ARE : BOOL := TRUE;
END_VAR
VAR_IN_OUT
	ARX : BOOL;
END_VAR
VAR_INPUT CONSTANT
	CYCLE_TIME : TIME;
	SENS : BYTE;
	SELF_ACT_TIME : TIME;
	SELF_ACT_PULSE : TIME;
	SELF_ACT_CYCLES : INT := 1;
END_VAR
VAR_OUTPUT
	OUT : BOOL;
	ARO : BOOL;
END_VAR
VAR
	timer : AUTORUN;
	pwgen : GEN_PULSE;
END_VAR


(*
version 2.1	24. jan. 2009
programmer 	hugo
tested by		oscat

this is an intelligent actuator interface for any 2point actuator like coil drive.
the 2Point actuator can only switch on/off and therefore the input must be converted to on/off cycles.
the interface can be programmed with double click on the symbol.
in addition a self_act_time and self_act_cycles ca be programmed to switch n times on/off every self_act_time to avoid a valve to freeze.
the input value must be between 0 and 255. with the setup variable sens one can specify what must be the minimum input to turn the valve on at all.
at the same time an input > 255-sens will turn the valve on at all times.


*)

(* run the autorun timer *)
timer(trun := SELF_ACT_PULSE * (2 * SELF_ACT_CYCLES), toff := SELF_ACT_TIME, Test := TEST, ARE := ARE, arx := ARX);
ARO := timer.ARO;

(* run the pulse width generator *)
IF aro THEN
	pwgen(PTL := SELF_ACT_PULSE, PTH := SELF_ACT_PULSE);
	out := pwgen.Q;
ELSIF in < sens THEN
	out := FALSE;
ELSIF in > BYTE#255 - sens THEN
	out := TRUE;
ELSE
	pwgen.PTH := (CYCLE_TIME * BAND_B(IN,SENS)) / 255;
	pwgen.PTL := CYCLE_TIME - pwgen.PTH;
	pwgen();
	out := pwgen.Q;
END_IF;



(* revision history
hm	7.10.2006 		rev 1.1
	changed error pos could not reach 1 or 0 under certain conditions due to error in code.
	changed on and off in force and force_in for better usability.

hm	17.1.2007		rev 1.2
	deleted unused variable time_overflow

hm	15.9.2007		rev 1.3
	replaced time() with T_PLC_MS for compatibility and performance reasons

hm	19. 11 2007		rev 1.4
	replaced left over statement time() with tx

hm	27. 12. 2007	REV 1.5
	CHANGED CODE FOR BETTER PERFORMANCE

hm	21. oct. 2008	rev 1.6
	code optimized

hm	23. nov. 2008	rev 2.0
	new code using library modules

hm	24. jan. 2009	rev 2.1
	deleted unused var inb
*)

END_FUNCTION_BLOCK

// POUs/Building/actuators/AUTORUN
FUNCTION_BLOCK AUTORUN
VAR_INPUT
	IN : BOOL;
	TEST : BOOL;
	ARE : BOOL := TRUE;
END_VAR
VAR_IN_OUT
	ARX : BOOL;
END_VAR
VAR_INPUT CONSTANT
	TRUN : TIME;
	TOFF : TIME;
END_VAR
VAR_OUTPUT
	OUT : BOOL;
	ARO : BOOL;
END_VAR
VAR
	timer : _RMP_B;
	val : BYTE;
END_VAR



(*
version 1.0	20. nov 2008
programmer 	hugo
tested by	oscat




*)

(* run the integrator when T_off > T#0s *)
IF TOFF > T#0s THEN
	timer(DIR:= OUT, TR := SEL(OUT, TOFF, TRUN), RMP := val);
ELSE
	val := 255;
END_IF;


(* when timer = 0 or test then initiate autorun until timer reaches 255 *)
IF (NOT ARX AND ARE AND val = 0) OR TEST THEN
	val := 0;
	ARO := TRUE;
	ARX := TRUE;
ELSIF val = 255 AND ARO THEN
	ARO := FALSE;
	ARX := FALSE;
END_IF;

(* output is true when autorun ARO is true or in = TRUE *)
out := IN OR ARO;



(* revision history
hm 20. nov. 2008	rev 1.0
	original version

*)

END_FUNCTION_BLOCK

// POUs/Engineering/measurements/CYCLE_TIME
FUNCTION_BLOCK CYCLE_TIME
VAR_INPUT
	RST : BOOL;
END_VAR
VAR_OUTPUT
	ct_min : TIME;
	ct_max : TIME;
	ct_last : TIME;
	systime : TIME;
	sysdays : INT;
	cycles : DWORD;
END_VAR
VAR
	last_cycle : TIME;
	tx: TIME;
	init: BOOL;
END_VAR


(*
	version 1.2	16 sep 2007
	programmer 	hugo
	tested BY		hans

this function block measures the cycle time and displays the last, min and max cycle time of the current task.
the resolution is 1ms.
the cycles output is a dword counter which counts the cycles.
a rst pulse on the input will reset all data.


*)

tx := DWORD_TO_TIME(T_PLC_MS()) - last_cycle;
IF rst THEN
	ct_min := t#10h;
	ct_max := t#0ms;
	cycles := 0;
ELSIF last_cycle > t#0s THEN
	IF tx < ct_min THEN ct_min := tx;
	ELSIF tx > ct_max THEN ct_max := tx;
	END_IF;
	ct_last := tx;
ELSIF ct_min = t#0s THEN
	ct_min := t#0s - t#1ms;
END_IF;
IF init THEN
	systime := systime + tx;
		IF systime >= t#1d THEN
			systime := systime - t#1d;
			sysdays := sysdays + 1;
		END_IF;
END_IF;
init := TRUE;
last_cycle := last_cycle + tx;
cycles := cycles + 1;

(*	revision history
hm 12.12.2006		rev 1.1
	added cycles output, a dword cycle counter.
hm 10.3.2007			rev 1.2
	changed initialization of ct_min to t#10h for compatibility with siemens s7

hm	16.9.2007		rev 1.2
	changed Time() in T_PLC_MS() for compatibility resons

*)

END_FUNCTION_BLOCK

// POUs/Engineering/control/BAND_B
FUNCTION BAND_B : BYTE
VAR_INPUT
	X : BYTE;
	B : BYTE;
END_VAR



(*
version 1.0	21. Nov. 2008
programmer 	hugo
tested by	oscat

BAND_B will limit X to B <= X <= 255-B. while X < B the resulkt will be 0 and while X > 255-B the output will be 255
otherwise the result = X.

*)

IF X < B THEN
	BAND_B := 0;
ELSIF X > BYTE#255-B THEN
	BAND_B := 255;
ELSE
	BAND_B := X;
END_IF;



(* revision history
hm	21. nov. 2008	rev 1.0
	original version

*)

END_FUNCTION

// POUs/Engineering/signal generators/GEN_PULSE
FUNCTION_BLOCK GEN_PULSE
VAR_INPUT
	ENQ : BOOL := TRUE;
	PTH : TIME;
	PTL : TIME;
END_VAR
VAR_OUTPUT
	Q : BOOL;
END_VAR
VAR
	tx: TIME;
	tn: TIME;
	init: BOOL;
END_VAR

(*
version 1.3	13. nov. 2009
programmer 	hugo
tested by		oscat

GEN_PULSE uses the internal sps timer to generate a continuous output waveform with programmable high and low time.
the accuracy of gen_pulse is depending on the system timer.
when time is 0 the high and low times are exactly one cycle.
ENQ = TRUE will start and ENQ = FALSE will stop the generator.

*)

(* read system timer *)
IF enq THEN
	tx := DWORD_TO_TIME(T_PLC_MS());
	IF NOT init THEN init := TRUE; tn := tx; END_IF;
	IF tx >= tn THEN
		Q := NOT Q;
		tn := tn + SEL(Q,PTL,PTH);
	END_IF;
ELSE
	Q := FALSE;
	init := FALSE;
END_IF;



(* revision history
hm	29. jun. 2008	rev 1.0
	original version

hm	23. nov. 2008	rev 1.1
	set default for enq to be true

hm	18. jul. 2009	rev 1.2
	improved performance

hm	13. nov. 2009	rev 1.3
	corrected error

*)

END_FUNCTION_BLOCK

// POUs/Building/electrical/CLICK
FUNCTION_BLOCK CLICK
VAR_INPUT
	in : BOOL;
END_VAR
VAR_OUTPUT
	Q : BOOL;
	single : BOOL;
	double : BOOL;
	triple : BOOL;
	status: BYTE;
END_VAR
VAR_INPUT CONSTANT
	T_debounce : TIME := t#10ms;
	T_short : TIME := t#200ms;
	T_pause : TIME := t#500ms;
	T_reconfig : TIME := t#1m;
END_VAR
VAR
	s_in : SW_RECONFIG;
	tx: TIME;
	state: INT;
	last: TIME;
END_VAR

(*
version 2.0	28. dec. 2008
programmer 	oscat
tested by		oscat

click checks an input for single, double or tripple click and sets the corresponding output single, doulbe or triple for the time the input stays high at the last click.
the maximum high and low time for a click can be configured with setup variables.
the input configures itself to be high or low active depending on which state the input stays longer than t_reconfig.

*)

(* reconfiguration and debounce circuitry *)
s_in(in := in, TD := T_debounce, TR := T_reconfig);

(* read system time *)
tx := DWORD_TO_TIME(T_PLC_MS());

(* count the mumber of clicks *)
IF s_in.Q XOR Q THEN
	last := tx;
	IF s_in.Q THEN state := state + 1; END_IF;
END_IF;
Q := s_in.Q;

(* set outputs *)
IF state > 0 THEN
	IF (Q AND tx - last > t_short) OR (NOT Q AND tx - last > t_pause) THEN
		CASE state OF
			1:	single := TRUE;
				status := 111;
			2:	double := TRUE;
				status := 112;
			3:	triple := TRUE;
				status := 113;
		END_CASE;
		state := 0;
	END_IF;
ELSIF NOT q THEN
	single := FALSE;
	double := FALSE;
	triple := FALSE;
	status := 110;
	last := tx;
	state := 0;
END_IF;





(* revision history

15 Feb 2007	rev 1.0	hm
	created original version

18.5.2007	rev 1.1 hm
	corrected an error while execution would stop after t_reconfig elapsed.

15.9.2007	rev 1.2 hm
	replaced Time() with T_PLC_MS for compatibility and performance reasons

28. dec. 2008	rev 2.0
	rewritten using modular approach

*)

END_FUNCTION_BLOCK

// POUs/Building/electrical/DEBOUNCE
FUNCTION_BLOCK DEBOUNCE
VAR_INPUT
	IN : BOOL;
	TD : TIME;
	PM : BOOL;
END_VAR

VAR_OUTPUT
	Q : BOOL;
END_VAR
VAR
	deb : TOF;
END_VAR

(*
version 1.0	22. sep. 2008
programmer 	oscat
tested by	tobias

DEBOUNCE is used to debounce switch inputs.
in addition to the debounce functionality this FB can also be used to detect rising edges on IN when PM = TRUE.
When PM = FALSE, Q follows in with the debounce functionality.

*)


IF NOT deb.Q AND IN THEN
	(* rising edge on input detetced a *)
	Q := TRUE;
ELSIF NOT PM THEN
	Q := deb.Q;
ELSE
	Q := FALSE;
END_IF;

(* run debounce timer *)
deb(IN := IN, PT := TD);



(*
hm 22. sep. 2008	rev 1.0
	original version

*)

END_FUNCTION_BLOCK

// POUs/Building/electrical/SW_RECONFIG
FUNCTION_BLOCK SW_RECONFIG
VAR_INPUT
	IN : BOOL;
	TD : TIME;
	TR : TIME;
END_VAR
VAR_OUTPUT
	Q : BOOL;
END_VAR
VAR
	T1, T2 : TON;
	INV: BOOL;
END_VAR


(*
version 1.0	22. oct. 2008
programmer 	hugo
tested by	oscat

SW_reconfig detects if an input is high or low active and debounces the input

*)

(* run debounce circuit *)
t1(in := IN, PT := TD);

IF tr > t#0s THEN
	(* generate output *)
	Q := t1.Q XOR inv;
	(* reconfiguration timer *)
	T2(in := Q, pt := TR);
	(* when T2.Q goes high then reverse INV *)
	IF T2.Q THEN INV := NOT INV; END_IF;
ELSE
	Q := t1.Q;
END_IF;



(* revision history
hm	22.10.2008	rev 1.0
	original version

*)

END_FUNCTION_BLOCK

// POUs/Mathematical/INV
FUNCTION INV : REAL
VAR_INPUT
	X : REAL;
END_VAR


(*
version 1.1	10. mar. 2009
programmer 	hugo
tested by		tobias

This function calculates the result of 1 / X

*)

IF X <> 0.0 THEN INV := 1.0 / X; END_IF;




(* revision history
hm	26. oct. 2008	rev 1.0
	original version

hm	10. mar. 2009	rev 1.1
	real constants updated to new systax using dot

*)

END_FUNCTION

// POUs/Logic/gate logic/REVERSE
FUNCTION REVERSE : BYTE
VAR_INPUT
	IN : BYTE;
END_VAR


(*
	version 1.1	18. feb 2008
	programmer 	hugo
	tested BY		tobias

This function reverses the bits of a byte so that after execution bit 7 is at bit 0 location and so forth.

*)

REVERSE := SHL(in,7) OR SHR(in,7) OR (ROR(in,3) AND 2#01000100) OR (ROL(in,3) AND 2#00100010)
	OR (SHL(in,1) AND 2#00010000) OR (SHR(in,1) AND 2#00001000);


(* revision history
hm		9.oct 2007		rev 1.0
	original version

hm		18. feb 2008	rev 1.1
	improved performance
*)

END_FUNCTION

// POUs/Building/actuators/ACTUATOR_3P
FUNCTION_BLOCK ACTUATOR_3P
VAR_INPUT
	in : REAL;
	force : BOOL;
	on : BOOL;
	end_pos : BOOL;
	diag : BOOL;
END_VAR
VAR_INPUT CONSTANT
	min_ontime : TIME := t#10s;
	min_offtime : TIME := t#10s;
	max_runtime : TIME := t#60s;
	auto_diag_time : TIME := t#10d;
	cal_runtime : TIME := t#600s;
	switch_available: BOOL;
END_VAR
VAR_OUTPUT
	out1 : BOOL;
	out2 : BOOL;
	pos : REAL;
	busy : BOOL;
	error : BOOL;
END_VAR
VAR
	val: REAL;
	tx : TIME;
	last_diag: TIME;
	last : TIME;
	runtime_1 : TIME;
	runtime_2 : TIME;
	state : INT;
	rout: FT_RMP;
	end : R_TRIG;
	cal_timer: TIME;
	Tn: TIME;
END_VAR


(*
version 1.3	 15 sep 2007
programmer 	hugo
tested by	oscat

actuator_3P is an interface for a 3 point actuator.
a 3P actuator is a motor with 2 directions that drives a valve or flap. the position of the valve or flap is controlled by runtime of the motor foreward or backward.
the available inputs are:
in is a real value which specifies the position of the actuator, 0 = 0% and 1 = 100% any value <0 or > 1 is limited to 0 or 1.
a force input must be low for normal operation and if switched high, the motor can only be controlled for 0% or 100% positions with the on input.
an and pos input is available for a end_pos switch, this switch indicates the valve or flap to be at either 0% or 100%
a diag input can at any time start a diag cycle which turns the motor towards the 0% position, then measures the runtime to 100% and then the runtime to 0%
these runtimes are stored and used for absolute positioning of the motor during normal operation.
a setup constand "auto_diag_time can be used to specify how often the actuator repeates this auto_diag cycla automatically.
at power on a cycle is perfomed automatically.
a 0 for this value means auto diag is never performed.

the outputs ar out1 and out2 for up and down direction of the motor. to avoid flickering the output can be programmed for min_ontime and min_offtime.
a pos outout indicates the absulute position of the actuator during operation and a busy output indicates the actuator is busy.
a error output is initiated when the specified max_runtime is reached by any direction during debug.
also when the up and down direction differs by more then 10% the error output is set.

for absolute positioning accuracy the actuator has a setup variable "cal_runtime" if this is set the actuator measures the total runtime of the motors and when this 
cal_runtime is exceeded it resets the actuator to 0% position and sets the output again to assure absolute accuracy.

autodiag and calibration can be shut off by setting the appropriate values to 0.
a switch_available setup variable specifies if end_pos switches are available.

*)

(* setup *)
Tn := DWORD_TO_TIME(T_PLC_MS());
tx := Tn - last;
end(clk := end_pos);

(* init only when first started *)
IF state = 0 THEN
	runtime_1 := max_runtime;
	runtime_2 := max_runtime;
	state := 1;
	rout(KR := 1000 / TIME_TO_REAL(runtime_1), KF := 1000 / TIME_TO_REAL(runtime_1) );
	tx := t#0s;
	last := Tn;
	last_diag := last;
END_IF;

(* check for end_sw and stop if reached *)
IF switch_available AND out1 AND end.Q THEN
	(* upper limit has been reached *)
	out1 := 0;
	rout(rmp := 0, in := 1);
	rout.Rmp := 1;
ELSIF switch_available AND out2 AND end.Q THEN
	(* lower limit has been reached *)
	out2 := 0;
	rout(rmp := 0, in := 0);
	rout.Rmp := 1;
END_IF;

(* check for min_offtime and min_ontime and return if it has not elapsed *)
IF NOT busy AND tx < min_offtime THEN
	RETURN;
ELSIF busy AND tx < min_ontime THEN
	RETURN;

(* check for last diag cycle and start diag if auto_diag_time has elapsed *)
ELSIF (tn - last_diag > auto_diag_time AND state > 10 AND auto_diag_time > t#0s) OR (diag AND state >= 10) THEN state := 1;

(* check if force pin is high *)
ELSIF force THEN state := 10;

(* check if calibration is necessary *)
ELSIF cal_timer > cal_runtime AND state = 99 AND cal_runtime > t#0s THEN state := 20;
END_IF;

(* state machine for operation *)
CASE state OF

